LIN {X 0,Y 312.481,Z 159.56,A -85,B 0,C 180,E1 -15787.929,E2 -15787.929} C_VEL
LIN {X 0,Y 311.791,Z 159.647,A -85,B 0,C 180,E1 -15789.004,E2 -15789.004} C_VEL
LIN {X 0,Y 308.912,Z 160.004,A -85,B 0,C 180,E1 -15790.755,E2 -15790.755} C_VEL
LIN {X 0,Y 306.5,Z 160.304,A -85,B 0,C 180,E1 -15792.174,E2 -15792.174} C_VEL
LIN {X 0,Y 305.491,Z 160.433,A -85,B 0,C 180,E1 -15793.274,E2 -15793.274} C_VEL
LIN {X 0,Y 305.422,Z 160.441,A -85,B 0,C 180,E1 -15793.646,E2 -15793.646} C_VEL
LIN {X 0,Y 305.436,Z 160.44,A -85,B 0,C 180,E1 -15797.418,E2 -15797.418} C_VEL
LIN {X 0,Y 305.46,Z 160.435,A -85,B 0,C 180,E1 -15801.595,E2 -15801.595} C_VEL
LIN {X 0,Y 305.461,Z 160.432,A -85,B 0,C 180,E1 -15804.886,E2 -15804.886} C_VEL
LIN {X 0,Y 305.441,Z 160.436,A -85,B 0,C 180,E1 -15808.358,E2 -15808.358} C_VEL
LIN {X 0,Y 305.475,Z 160.43,A -85,B 0,C 180,E1 -15811.109,E2 -15811.109} C_VEL
LIN {X 0,Y 305.5,Z 160.429,A -85,B 0,C 180,E1 -15814.081,E2 -15814.081} C_VEL
LIN {X 0,Y 305.484,Z 160.426,A -85,B 0,C 180,E1 -15818.402,E2 -15818.402} C_VEL
LIN {X 0,Y 305.508,Z 160.428,A -85,B 0,C 180,E1 -15821.212,E2 -15821.212} C_VEL
LIN {X 0,Y 305.578,Z 160.412,A -85,B 0,C 180,E1 -15825.345,E2 -15825.345} C_VEL
LIN {X 0,Y 305.623,Z 160.413,A -85,B 0,C 180,E1 -15829.399,E2 -15829.399} C_VEL
LIN {X 0,Y 305.744,Z 160.396,A -85,B 0,C 180,E1 -15832.072,E2 -15832.072} C_VEL
LIN {X 0,Y 305.653,Z 160.409,A -85,B 0,C 180,E1 -15834.723,E2 -15834.723} C_VEL
LIN {X 0,Y 305.933,Z 160.373,A -85,B 0,C 180,E1 -15838.684,E2 -15838.684} C_VEL
LIN {X 0,Y 305.931,Z 160.366,A -85,B 0,C 180,E1 -15841.316,E2 -15841.316} C_VEL
LIN {X 0,Y 305.783,Z 160.392,A -85,B 0,C 180,E1 -15846.599,E2 -15846.599} C_VEL
LIN {X 0,Y 305.682,Z 160.4,A -85,B 0,C 180,E1 -15849.261,E2 -15849.261} C_VEL
LIN {X 0,Y 305.551,Z 160.423,A -85,B 0,C 180,E1 -15853.298,E2 -15853.298} C_VEL
LIN {X 0,Y 305.49,Z 160.424,A -85,B 0,C 180,E1 -15856.026,E2 -15856.026} C_VEL
LIN {X 0,Y 305.471,Z 160.432,A -85,B 0,C 180,E1 -15860.188,E2 -15860.188} C_VEL
LIN {X 0,Y 305.438,Z 160.434,A -85,B 0,C 180,E1 -15864.467,E2 -15864.467} C_VEL
LIN {X 0,Y 305.447,Z 160.437,A -85,B 0,C 180,E1 -15867.399,E2 -15867.399} C_VEL
LIN {X 0,Y 305.428,Z 160.436,A -85,B 0,C 180,E1 -15870.413,E2 -15870.413} C_VEL
LIN {X 0,Y 305.464,Z 160.429,A -85,B 0,C 180,E1 -15874.078,E2 -15874.078} C_VEL
LIN {X 0,Y 305.453,Z 160.437,A -85,B 0,C 180,E1 -15876.743,E2 -15876.743} C_VEL
LIN {X 0,Y 305.409,Z 160.442,A -85,B 0,C 180,E1 -15880.59,E2 -15880.59} C_VEL
LIN {X 0,Y 305.421,Z 160.438,A -85,B 0,C 180,E1 -15883.656,E2 -15883.656} C_VEL
LIN {X 0,Y 305.434,Z 160.436,A -85,B 0,C 180,E1 -15887.419,E2 -15887.419} C_VEL
LIN {X 0,Y 305.461,Z 160.433,A -85,B 0,C 180,E1 -15891.595,E2 -15891.595} C_VEL
LIN {X 0,Y 305.463,Z 160.437,A -85,B 0,C 180,E1 -15894.887,E2 -15894.887} C_VEL
LIN {X 0,Y 305.485,Z 160.457,A -85,B 0,C 180,E1 -15896.205,E2 -15896.205} C_VEL
LIN {X 0,Y 308.142,Z 171.998,A -85,B 0,C 180,E1 -15899.883,E2 -15899.883} C_VEL
LIN {X 0,Y 309.87,Z 180.598,A -85,B 0,C 180,E1 -15902.483,E2 -15902.483} C_VEL
LIN {X 0,Y 310.416,Z 185.1,A -85,B 0,C 180,E1 -15903.78,E2 -15903.78} C_VEL
LIN {X 0,Y 315.255,Z 212.189,A -85,B 0,C 180,E1 -15904.876,E2 -15904.876} C_VEL
LIN {X 0,Y 317.606,Z 229.16,A -85,B 0,C 180,E1 -15905.486,E2 -15905.486} C_VEL
LIN {X 0,Y 316.044,Z 293.949,A -85,B 0,C 180,E1 -15906.968,E2 -15906.968} C_VEL
LIN {X 0,Y 315.164,Z 307.123,A -85,B 0,C 180,E1 -15907.506,E2 -15907.506} C_VEL
LIN {X 0,Y 313.89,Z 320.349,A -85,B 0,C 180,E1 -15908.319,E2 -15908.319} C_VEL
LIN {X 0,Y 312.567,Z 331.466,A -85,B 0,C 180,E1 -15909.259,E2 -15909.259} C_VEL
LIN {X 0,Y 311.014,Z 343.05,A -85,B 0,C 180,E1 -15910.53,E2 -15910.53} C_VEL
LIN {X 0,Y 309.393,Z 353.483,A -85,B 0,C 180,E1 -15911.971,E2 -15911.971} C_VEL
LIN {X 0,Y 308.101,Z 362.46,A -85,B 0,C 180,E1 -15913.517,E2 -15913.517} C_VEL
LIN {X 0,Y 306.676,Z 371.281,A -85,B 0,C 180,E1 -15915.399,E2 -15915.399} C_VEL
LIN {X 0,Y 305.431,Z 378.722,A -85,B 0,C 180,E1 -15917.373,E2 -15917.373} C_VEL
LIN {X 0,Y 304.614,Z 384.707,A -85,B 0,C 180,E1 -15919.363,E2 -15919.363} C_VEL
LIN {X 0,Y 304.052,Z 389.439,A -85,B 0,C 180,E1 -15921.358,E2 -15921.358} C_VEL
LIN {X 0,Y 303.72,Z 393.058,A -85,B 0,C 180,E1 -15923.355,E2 -15923.355} C_VEL
LIN {X 0,Y 303.638,Z 394.926,A -85,B 0,C 180,E1 -15924.687,E2 -15924.687} C_VEL
LIN {X 0,Y 303.629,Z 396.329,A -85,B 0,C 180,E1 -15926.018,E2 -15926.018} C_VEL
LIN {X 0,Y 303.624,Z 397.33,A -85,B 0,C 180,E1 -15927.346,E2 -15927.346} C_VEL
LIN {X 0,Y 303.614,Z 397.94,A -85,B 0,C 180,E1 -15928.673,E2 -15928.673} C_VEL
LIN {X 0,Y 303.667,Z 398.156,A -85,B 0,C 180,E1 -15929.999,E2 -15929.999} C_VEL
LIN {X 0,Y 303.614,Z 397.933,A -85,B 0,C 180,E1 -15931.326,E2 -15931.326} C_VEL
LIN {X 0,Y 303.624,Z 397.319,A -85,B 0,C 180,E1 -15932.653,E2 -15932.653} C_VEL
LIN {X 0,Y 303.63,Z 396.314,A -85,B 0,C 180,E1 -15933.981,E2 -15933.981} C_VEL
LIN {X 0,Y 303.625,Z 394.595,A -85,B 0,C 180,E1 -15935.544,E2 -15935.544} C_VEL
LIN {X 0,Y 303.943,Z 390.715,A -85,B 0,C 180,E1 -15937.974,E2 -15937.974} C_VEL
LIN {X 0,Y 304.383,Z 386.352,A -85,B 0,C 180,E1 -15939.971,E2 -15939.971} C_VEL
LIN {X 0,Y 305.092,Z 380.8,A -85,B 0,C 180,E1 -15941.964,E2 -15941.964} C_VEL
LIN {X 0,Y 306.255,Z 373.882,A -85,B 0,C 180,E1 -15943.942,E2 -15943.942} C_VEL
LIN {X 0,Y 307.655,Z 365.226,A -85,B 0,C 180,E1 -15945.909,E2 -15945.909} C_VEL
LIN {X 0,Y 308.931,Z 356.351,A -85,B 0,C 180,E1 -15947.543,E2 -15947.543} C_VEL
LIN {X 0,Y 310.58,Z 345.437,A -85,B 0,C 180,E1 -15949.153,E2 -15949.153} C_VEL
LIN {X 0,Y 312.132,Z 334.421,A -85,B 0,C 180,E1 -15950.425,E2 -15950.425} C_VEL
LIN {X 0,Y 313.617,Z 322.074,A -85,B 0,C 180,E1 -15951.527,E2 -15951.527} C_VEL
LIN {X 0,Y 314.804,Z 310.379,A -85,B 0,C 180,E1 -15952.303,E2 -15952.303} C_VEL
LIN {X 0,Y 315.802,Z 297.871,A -85,B 0,C 180,E1 -15952.876,E2 -15952.876} C_VEL
LIN {X 0,Y 316.354,Z 281.908,A -85,B 0,C 180,E1 -15953.31,E2 -15953.31} C_VEL
LIN {X 0,Y 317.411,Z 226.976,A -85,B 0,C 180,E1 -15954.557,E2 -15954.557} C_VEL
LIN {X 0,Y 312.684,Z 197.182,A -85,B 0,C 180,E1 -15955.688,E2 -15955.688} C_VEL
LIN {X 0,Y 310.379,Z 185.064,A -85,B 0,C 180,E1 -15956.202,E2 -15956.202} C_VEL
LIN {X 0,Y 309.526,Z 178.852,A -85,B 0,C 180,E1 -15958.008,E2 -15958.008} C_VEL
LIN {X 0,Y 307.186,Z 167.923,A -85,B 0,C 180,E1 -15961.364,E2 -15961.364} C_VEL
LIN {X 0,Y 305.481,Z 160.432,A -85,B 0,C 180,E1 -15963.794,E2 -15963.794} C_VEL
LIN {X 0,Y 305.45,Z 160.429,A -85,B 0,C 180,E1 -15966.741,E2 -15966.741} C_VEL
LIN {X 0,Y 305.405,Z 160.439,A -85,B 0,C 180,E1 -15970.589,E2 -15970.589} C_VEL
LIN {X 0,Y 305.416,Z 160.441,A -85,B 0,C 180,E1 -15973.655,E2 -15973.655} C_VEL
LIN {X 0,Y 305.43,Z 160.441,A -85,B 0,C 180,E1 -15977.417,E2 -15977.417} C_VEL
LIN {X 0,Y 305.454,Z 160.435,A -85,B 0,C 180,E1 -15981.594,E2 -15981.594} C_VEL
LIN {X 0,Y 305.455,Z 160.438,A -85,B 0,C 180,E1 -15984.886,E2 -15984.886} C_VEL
LIN {X 0,Y 305.435,Z 160.435,A -85,B 0,C 180,E1 -15988.357,E2 -15988.357} C_VEL
LIN {X 0,Y 305.468,Z 160.429,A -85,B 0,C 180,E1 -15991.108,E2 -15991.108} C_VEL
LIN {X 0,Y 305.473,Z 160.431,A -85,B 0,C 180,E1 -15994.079,E2 -15994.079} C_VEL
LIN {X 0,Y 305.45,Z 160.434,A -85,B 0,C 180,E1 -15998.399,E2 -15998.399} C_VEL
LIN {X 0,Y 305.494,Z 160.429,A -85,B 0,C 180,E1 -16001.212,E2 -16001.212} C_VEL
LIN {X 0,Y 305.57,Z 160.418,A -85,B 0,C 180,E1 -16005.345,E2 -16005.345} C_VEL
LIN {X 0,Y 305.614,Z 160.411,A -85,B 0,C 180,E1 -16009.399,E2 -16009.399} C_VEL
LIN {X 0,Y 305.729,Z 160.4,A -85,B 0,C 180,E1 -16012.072,E2 -16012.072} C_VEL
LIN {X 0,Y 305.645,Z 160.41,A -85,B 0,C 180,E1 -16014.723,E2 -16014.723} C_VEL
LIN {X 0,Y 305.924,Z 160.373,A -85,B 0,C 180,E1 -16018.684,E2 -16018.684} C_VEL
LIN {X 0,Y 305.926,Z 160.376,A -85,B 0,C 180,E1 -16021.316,E2 -16021.316} C_VEL
LIN {X 0,Y 305.777,Z 160.392,A -85,B 0,C 180,E1 -16026.599,E2 -16026.599} C_VEL
LIN {X 0,Y 305.686,Z 160.407,A -85,B 0,C 180,E1 -16029.261,E2 -16029.261} C_VEL
LIN {X 0,Y 305.563,Z 160.416,A -85,B 0,C 180,E1 -16033.297,E2 -16033.297} C_VEL
LIN {X 0,Y 305.505,Z 160.429,A -85,B 0,C 180,E1 -16036.025,E2 -16036.025} C_VEL
LIN {X 0,Y 305.478,Z 160.428,A -85,B 0,C 180,E1 -16040.188,E2 -16040.188} C_VEL
LIN {X 0,Y 305.479,Z 160.433,A -85,B 0,C 180,E1 -16043.04,E2 -16043.04} C_VEL
LIN {X 0,Y 305.446,Z 160.43,A -85,B 0,C 180,E1 -16046.191,E2 -16046.191} C_VEL
LIN {X 0,Y 305.442,Z 160.439,A -85,B 0,C 180,E1 -16049.034,E2 -16049.034} C_VEL
LIN {X 0,Y 305.43,Z 160.434,A -85,B 0,C 180,E1 -16051.954,E2 -16051.954} C_VEL
LIN {X 0,Y 305.455,Z 160.437,A -85,B 0,C 180,E1 -16055.114,E2 -16055.114} C_VEL
LIN {X 0,Y 305.427,Z 160.439,A -85,B 0,C 180,E1 -16058.526,E2 -16058.526} C_VEL
LIN {X 0,Y 305.431,Z 160.44,A -85,B 0,C 180,E1 -16062.583,E2 -16062.583} C_VEL
LIN {X 0,Y 305.418,Z 160.439,A -85,B 0,C 180,E1 -16066.345,E2 -16066.345} C_VEL
LIN {X 0,Y 305.454,Z 160.435,A -85,B 0,C 180,E1 -16069.893,E2 -16069.893} C_VEL
LIN {X 0,Y 305.46,Z 160.434,A -85,B 0,C 180,E1 -16073.637,E2 -16073.637} C_VEL
LIN {X 0,Y 305.463,Z 160.438,A -85,B 0,C 180,E1 -16076.484,E2 -16076.484} C_VEL
LIN {X 0,Y 305.429,Z 160.437,A -85,B 0,C 180,E1 -16079.589,E2 -16079.589} C_VEL
LIN {X 0,Y 305.527,Z 160.543,A -85,B 0,C 180,E1 -16081.912,E2 -16081.912} C_VEL
LIN {X 0,Y 306.578,Z 165.2,A -85,B 0,C 180,E1 -16083.493,E2 -16083.493} C_VEL
LIN {X 0,Y 314.759,Z 184.793,A -85,B 0,C 180,E1 -16084.743,E2 -16084.743} C_VEL
LIN {X 0,Y 317.517,Z 192.242,A -85,B 0,C 180,E1 -16085.163,E2 -16085.163} C_VEL
LIN {X 0,Y 318.252,Z 196.661,A -85,B 0,C 180,E1 -16085.333,E2 -16085.333} C_VEL
LIN {X 0,Y 316.461,Z 271.983,A -85,B 0,C 180,E1 -16087.045,E2 -16087.045} C_VEL
LIN {X 0,Y 315.766,Z 285.365,A -85,B 0,C 180,E1 -16087.596,E2 -16087.596} C_VEL
LIN {X 0,Y 314.898,Z 296.992,A -85,B 0,C 180,E1 -16088.307,E2 -16088.307} C_VEL
LIN {X 0,Y 313.577,Z 309.444,A -85,B 0,C 180,E1 -16089.33,E2 -16089.33} C_VEL
LIN {X 0,Y 312.107,Z 321.083,A -85,B 0,C 180,E1 -16090.603,E2 -16090.603} C_VEL
LIN {X 0,Y 310.863,Z 331.53,A -85,B 0,C 180,E1 -16092.063,E2 -16092.063} C_VEL
LIN {X 0,Y 309.504,Z 340.047,A -85,B 0,C 180,E1 -16093.511,E2 -16093.511} C_VEL
LIN {X 0,Y 308.172,Z 347.905,A -85,B 0,C 180,E1 -16095.135,E2 -16095.135} C_VEL
LIN {X 0,Y 306.815,Z 355.583,A -85,B 0,C 180,E1 -16097.096,E2 -16097.096} C_VEL
LIN {X 0,Y 305.606,Z 362.627,A -85,B 0,C 180,E1 -16099.399,E2 -16099.399} C_VEL
LIN {X 0,Y 304.855,Z 367.315,A -85,B 0,C 180,E1 -16101.383,E2 -16101.383} C_VEL
LIN {X 0,Y 304.369,Z 370.9,A -85,B 0,C 180,E1 -16103.371,E2 -16103.371} C_VEL
LIN {X 0,Y 304.151,Z 372.752,A -85,B 0,C 180,E1 -16104.697,E2 -16104.697} C_VEL
LIN {X 0,Y 303.94,Z 374.146,A -85,B 0,C 180,E1 -16106.023,E2 -16106.023} C_VEL
LIN {X 0,Y 303.684,Z 375.749,A -85,B 0,C 180,E1 -16108.675,E2 -16108.675} C_VEL
LIN {X 0,Y 303.678,Z 375.979,A -85,B 0,C 180,E1 -16110.001,E2 -16110.001} C_VEL
LIN {X 0,Y 303.683,Z 375.788,A -85,B 0,C 180,E1 -16111.327,E2 -16111.327} C_VEL
LIN {X 0,Y 303.934,Z 374.237,A -85,B 0,C 180,E1 -16113.978,E2 -16113.978} C_VEL
LIN {X 0,Y 304.128,Z 372.883,A -85,B 0,C 180,E1 -16115.304,E2 -16115.304} C_VEL
LIN {X 0,Y 304.472,Z 370.494,A -85,B 0,C 180,E1 -16116.995,E2 -16116.995} C_VEL
LIN {X 0,Y 305.006,Z 366.145,A -85,B 0,C 180,E1 -16119.283,E2 -16119.283} C_VEL
LIN {X 0,Y 305.917,Z 361.133,A -85,B 0,C 180,E1 -16121.261,E2 -16121.261} C_VEL
LIN {X 0,Y 306.998,Z 354.824,A -85,B 0,C 180,E1 -16123.234,E2 -16123.234} C_VEL
LIN {X 0,Y 308.313,Z 346.926,A -85,B 0,C 180,E1 -16125.198,E2 -16125.198} C_VEL
LIN {X 0,Y 310.034,Z 337.093,A -85,B 0,C 180,E1 -16127.139,E2 -16127.139} C_VEL
LIN {X 0,Y 311.47,Z 326.779,A -85,B 0,C 180,E1 -16128.756,E2 -16128.756} C_VEL
LIN {X 0,Y 312.826,Z 316.549,A -85,B 0,C 180,E1 -16130.036,E2 -16130.036} C_VEL
LIN {X 0,Y 314.139,Z 305.354,A -85,B 0,C 180,E1 -16131.147,E2 -16131.147} C_VEL
LIN {X 0,Y 315.314,Z 292.729,A -85,B 0,C 180,E1 -16132.094,E2 -16132.094} C_VEL
LIN {X 0,Y 316.136,Z 280.065,A -85,B 0,C 180,E1 -16132.766,E2 -16132.766} C_VEL
LIN {X 0,Y 316.79,Z 267.014,A -85,B 0,C 180,E1 -16133.191,E2 -16133.191} C_VEL
LIN {X 0,Y 318.32,Z 196.121,A -85,B 0,C 180,E1 -16134.791,E2 -16134.791} C_VEL
LIN {X 0,Y 316.871,Z 190.339,A -85,B 0,C 180,E1 -16135.055,E2 -16135.055} C_VEL
LIN {X 0,Y 309.139,Z 171.149,A -85,B 0,C 180,E1 -16136.221,E2 -16136.221} C_VEL
LIN {X 0,Y 306.606,Z 165.204,A -85,B 0,C 180,E1 -16136.625,E2 -16136.625} C_VEL
LIN {X 0,Y 305.495,Z 160.433,A -85,B 0,C 180,E1 -16138.326,E2 -16138.326} C_VEL
LIN {X 0,Y 305.439,Z 160.435,A -85,B 0,C 180,E1 -16141.953,E2 -16141.953} C_VEL
LIN {X 0,Y 305.464,Z 160.434,A -85,B 0,C 180,E1 -16145.113,E2 -16145.113} C_VEL
LIN {X 0,Y 305.421,Z 160.438,A -85,B 0,C 180,E1 -16148.522,E2 -16148.522} C_VEL
LIN {X 0,Y 305.436,Z 160.437,A -85,B 0,C 180,E1 -16152.582,E2 -16152.582} C_VEL
LIN {X 0,Y 305.422,Z 160.441,A -85,B 0,C 180,E1 -16153.646,E2 -16153.646} C_VEL
LIN {X 0,Y 304.783,Z 160.528,A -85,B 0,C 180,E1 -16154.746,E2 -16154.746} C_VEL
LIN {X 0,Y 301.917,Z 160.887,A -85,B 0,C 180,E1 -16156.535,E2 -16156.535} C_VEL
LIN {X 0,Y 299.467,Z 161.186,A -85,B 0,C 180,E1 -16157.987,E2 -16157.987} C_VEL
LIN {X 0,Y 298.416,Z 161.311,A -85,B 0,C 180,E1 -16159.113,E2 -16159.113} C_VEL
LIN {X 0,Y 298.332,Z 161.318,A -85,B 0,C 180,E1 -16159.494,E2 -16159.494} C_VEL
LIN {X 0,Y 298.427,Z 161.311,A -85,B 0,C 180,E1 -16163.197,E2 -16163.197} C_VEL
LIN {X 0,Y 298.393,Z 161.317,A -85,B 0,C 180,E1 -16167.199,E2 -16167.199} C_VEL
LIN {X 0,Y 298.402,Z 161.31,A -85,B 0,C 180,E1 -16170.625,E2 -16170.625} C_VEL
LIN {X 0,Y 298.445,Z 161.309,A -85,B 0,C 180,E1 -16174.92,E2 -16174.92} C_VEL
LIN {X 0,Y 298.42,Z 161.303,A -85,B 0,C 180,E1 -16177.864,E2 -16177.864} C_VEL
LIN {X 0,Y 298.473,Z 161.308,A -85,B 0,C 180,E1 -16180.752,E2 -16180.752} C_VEL
LIN {X 0,Y 298.509,Z 161.293,A -85,B 0,C 180,E1 -16184.99,E2 -16184.99} C_VEL
LIN {X 0,Y 298.581,Z 161.29,A -85,B 0,C 180,E1 -16189.146,E2 -16189.146} C_VEL
LIN {X 0,Y 298.696,Z 161.274,A -85,B 0,C 180,E1 -16191.884,E2 -16191.884} C_VEL
LIN {X 0,Y 298.623,Z 161.285,A -85,B 0,C 180,E1 -16194.598,E2 -16194.598} C_VEL
LIN {X 0,Y 298.901,Z 161.249,A -85,B 0,C 180,E1 -16198.653,E2 -16198.653} C_VEL
LIN {X 0,Y 298.899,Z 161.242,A -85,B 0,C 180,E1 -16201.347,E2 -16201.347} C_VEL
LIN {X 0,Y 298.731,Z 161.27,A -85,B 0,C 180,E1 -16206.755,E2 -16206.755} C_VEL
LIN {X 0,Y 298.614,Z 161.28,A -85,B 0,C 180,E1 -16209.483,E2 -16209.483} C_VEL
LIN {X 0,Y 298.506,Z 161.303,A -85,B 0,C 180,E1 -16213.618,E2 -16213.618} C_VEL
LIN {X 0,Y 298.428,Z 161.301,A -85,B 0,C 180,E1 -16216.416,E2 -16216.416} C_VEL
LIN {X 0,Y 298.427,Z 161.313,A -85,B 0,C 180,E1 -16219.609,E2 -16219.609} C_VEL
LIN {X 0,Y 298.381,Z 161.313,A -85,B 0,C 180,E1 -16223.604,E2 -16223.604} C_VEL
LIN {X 0,Y 298.401,Z 161.313,A -85,B 0,C 180,E1 -16226.583,E2 -16226.583} C_VEL
LIN {X 0,Y 298.391,Z 161.314,A -85,B 0,C 180,E1 -16229.644,E2 -16229.644} C_VEL
LIN {X 0,Y 298.392,Z 161.316,A -85,B 0,C 180,E1 -16232.801,E2 -16232.801} C_VEL
LIN {X 0,Y 298.427,Z 161.313,A -85,B 0,C 180,E1 -16236.802,E2 -16236.802} C_VEL
LIN {X 0,Y 298.373,Z 161.318,A -85,B 0,C 180,E1 -16239.492,E2 -16239.492} C_VEL
LIN {X 0,Y 298.37,Z 161.32,A -85,B 0,C 180,E1 -16243.097,E2 -16243.097} C_VEL
LIN {X 0,Y 298.37,Z 161.318,A -85,B 0,C 180,E1 -16246.915,E2 -16246.915} C_VEL
LIN {X 0,Y 298.385,Z 161.316,A -85,B 0,C 180,E1 -16251.011,E2 -16251.011} C_VEL
LIN {X 0,Y 298.406,Z 161.314,A -85,B 0,C 180,E1 -16253.928,E2 -16253.928} C_VEL
LIN {X 0,Y 298.463,Z 161.508,A -85,B 0,C 180,E1 -16255.716,E2 -16255.716} C_VEL
LIN {X 0,Y 300.842,Z 171.699,A -85,B 0,C 180,E1 -16259.073,E2 -16259.073} C_VEL
LIN {X 0,Y 302.701,Z 180.807,A -85,B 0,C 180,E1 -16261.918,E2 -16261.918} C_VEL
LIN {X 0,Y 303.392,Z 184.77,A -85,B 0,C 180,E1 -16263.115,E2 -16263.115} C_VEL
LIN {X 0,Y 305.029,Z 191.285,A -85,B 0,C 180,E1 -16263.445,E2 -16263.445} C_VEL
LIN {X 0,Y 309.487,Z 217.498,A -85,B 0,C 180,E1 -16264.513,E2 -16264.513} C_VEL
LIN {X 0,Y 311.149,Z 229.779,A -85,B 0,C 180,E1 -16264.964,E2 -16264.964} C_VEL
LIN {X 0,Y 309.542,Z 293.704,A -85,B 0,C 180,E1 -16266.455,E2 -16266.455} C_VEL
LIN {X 0,Y 308.564,Z 307.636,A -85,B 0,C 180,E1 -16267.042,E2 -16267.042} C_VEL
LIN {X 0,Y 307.286,Z 320.096,A -85,B 0,C 180,E1 -16267.828,E2 -16267.828} C_VEL
LIN {X 0,Y 305.932,Z 331.211,A -85,B 0,C 180,E1 -16268.788,E2 -16268.788} C_VEL
LIN {X 0,Y 304.305,Z 342.794,A -85,B 0,C 180,E1 -16270.083,E2 -16270.083} C_VEL
LIN {X 0,Y 302.61,Z 353.225,A -85,B 0,C 180,E1 -16271.552,E2 -16271.552} C_VEL
LIN {X 0,Y 301.147,Z 362.926,A -85,B 0,C 180,E1 -16273.278,E2 -16273.278} C_VEL
LIN {X 0,Y 299.761,Z 371.022,A -85,B 0,C 180,E1 -16275.054,E2 -16275.054} C_VEL
LIN {X 0,Y 298.487,Z 378.464,A -85,B 0,C 180,E1 -16277.074,E2 -16277.074} C_VEL
LIN {X 0,Y 297.614,Z 384.448,A -85,B 0,C 180,E1 -16279.11,E2 -16279.11} C_VEL
LIN {X 0,Y 297.008,Z 389.18,A -85,B 0,C 180,E1 -16281.152,E2 -16281.152} C_VEL
LIN {X 0,Y 296.645,Z 392.799,A -85,B 0,C 180,E1 -16283.196,E2 -16283.196} C_VEL
LIN {X 0,Y 296.552,Z 394.667,A -85,B 0,C 180,E1 -16284.56,E2 -16284.56} C_VEL
LIN {X 0,Y 296.527,Z 396.07,A -85,B 0,C 180,E1 -16285.922,E2 -16285.922} C_VEL
LIN {X 0,Y 296.548,Z 397.072,A -85,B 0,C 180,E1 -16287.283,E2 -16287.283} C_VEL
LIN {X 0,Y 296.531,Z 397.682,A -85,B 0,C 180,E1 -16288.641,E2 -16288.641} C_VEL
LIN {X 0,Y 296.579,Z 397.898,A -85,B 0,C 180,E1 -16289.999,E2 -16289.999} C_VEL
LIN {X 0,Y 296.531,Z 397.674,A -85,B 0,C 180,E1 -16291.357,E2 -16291.357} C_VEL
LIN {X 0,Y 296.549,Z 397.06,A -85,B 0,C 180,E1 -16292.716,E2 -16292.716} C_VEL
LIN {X 0,Y 296.527,Z 396.054,A -85,B 0,C 180,E1 -16294.077,E2 -16294.077} C_VEL
LIN {X 0,Y 296.546,Z 394.558,A -85,B 0,C 180,E1 -16295.508,E2 -16295.508} C_VEL
LIN {X 0,Y 296.782,Z 391.689,A -85,B 0,C 180,E1 -16297.483,E2 -16297.483} C_VEL
LIN {X 0,Y 297.19,Z 387.693,A -85,B 0,C 180,E1 -16299.528,E2 -16299.528} C_VEL
LIN {X 0,Y 297.957,Z 381.553,A -85,B 0,C 180,E1 -16301.91,E2 -16301.91} C_VEL
LIN {X 0,Y 299.106,Z 374.858,A -85,B 0,C 180,E1 -16303.935,E2 -16303.935} C_VEL
LIN {X 0,Y 300.535,Z 366.557,A -85,B 0,C 180,E1 -16305.948,E2 -16305.948} C_VEL
LIN {X 0,Y 301.85,Z 358.043,A -85,B 0,C 180,E1 -16307.618,E2 -16307.618} C_VEL
LIN {X 0,Y 303.475,Z 347.531,A -85,B 0,C 180,E1 -16309.268,E2 -16309.268} C_VEL
LIN {X 0,Y 305.275,Z 335.707,A -85,B 0,C 180,E1 -16310.729,E2 -16310.729} C_VEL
LIN {X 0,Y 306.796,Z 323.801,A -85,B 0,C 180,E1 -16311.853,E2 -16311.853} C_VEL
LIN {X 0,Y 308.123,Z 311.414,A -85,B 0,C 180,E1 -16312.725,E2 -16312.725} C_VEL
LIN {X 0,Y 309.218,Z 298.669,A -85,B 0,C 180,E1 -16313.347,E2 -16313.347} C_VEL
LIN {X 0,Y 309.786,Z 285.21,A -85,B 0,C 180,E1 -16313.745,E2 -16313.745} C_VEL
LIN {X 0,Y 310.961,Z 228.075,A -85,B 0,C 180,E1 -16315.067,E2 -16315.067} C_VEL
LIN {X 0,Y 306.443,Z 199.125,A -85,B 0,C 180,E1 -16316.194,E2 -16316.194} C_VEL
LIN {X 0,Y 303.978,Z 186.837,A -85,B 0,C 180,E1 -16316.738,E2 -16316.738} C_VEL
LIN {X 0,Y 303.38,Z 184.674,A -85,B 0,C 180,E1 -16316.884,E2 -16316.884} C_VEL
LIN {X 0,Y 301.58,Z 175.207,A -85,B 0,C 180,E1 -16319.785,E2 -16319.785} C_VEL
LIN {X 0,Y 298.973,Z 163.637,A -85,B 0,C 180,E1 -16323.532,E2 -16323.532} C_VEL
LIN {X 0,Y 298.423,Z 161.31,A -85,B 0,C 180,E1 -16324.363,E2 -16324.363} C_VEL
LIN {X 0,Y 298.394,Z 161.309,A -85,B 0,C 180,E1 -16327.76,E2 -16327.76} C_VEL
LIN {X 0,Y 298.343,Z 161.321,A -85,B 0,C 180,E1 -16331.267,E2 -16331.267} C_VEL
LIN {X 0,Y 298.35,Z 161.323,A -85,B 0,C 180,E1 -16335.034,E2 -16335.034} C_VEL
LIN {X 0,Y 298.343,Z 161.323,A -85,B 0,C 180,E1 -16338.92,E2 -16338.92} C_VEL
LIN {X 0,Y 298.391,Z 161.314,A -85,B 0,C 180,E1 -16342.238,E2 -16342.238} C_VEL
LIN {X 0,Y 298.401,Z 161.312,A -85,B 0,C 180,E1 -16345.58,E2 -16345.58} C_VEL
LIN {X 0,Y 298.37,Z 161.319,A -85,B 0,C 180,E1 -16348.788,E2 -16348.788} C_VEL
LIN {X 0,Y 298.403,Z 161.306,A -85,B 0,C 180,E1 -16351.898,E2 -16351.898} C_VEL
LIN {X 0,Y 298.406,Z 161.313,A -85,B 0,C 180,E1 -16354.917,E2 -16354.917} C_VEL
LIN {X 0,Y 298.382,Z 161.31,A -85,B 0,C 180,E1 -16357.861,E2 -16357.861} C_VEL
LIN {X 0,Y 298.445,Z 161.309,A -85,B 0,C 180,E1 -16360.751,E2 -16360.751} C_VEL
LIN {X 0,Y 298.502,Z 161.3,A -85,B 0,C 180,E1 -16364.99,E2 -16364.99} C_VEL
LIN {X 0,Y 298.572,Z 161.287,A -85,B 0,C 180,E1 -16369.146,E2 -16369.146} C_VEL
LIN {X 0,Y 298.675,Z 161.277,A -85,B 0,C 180,E1 -16371.884,E2 -16371.884} C_VEL
LIN {X 0,Y 298.616,Z 161.286,A -85,B 0,C 180,E1 -16374.598,E2 -16374.598} C_VEL
LIN {X 0,Y 298.892,Z 161.249,A -85,B 0,C 180,E1 -16378.653,E2 -16378.653} C_VEL
LIN {X 0,Y 298.894,Z 161.252,A -85,B 0,C 180,E1 -16381.347,E2 -16381.347} C_VEL
LIN {X 0,Y 298.726,Z 161.27,A -85,B 0,C 180,E1 -16386.756,E2 -16386.756} C_VEL
LIN {X 0,Y 298.618,Z 161.289,A -85,B 0,C 180,E1 -16389.483,E2 -16389.483} C_VEL
LIN {X 0,Y 298.515,Z 161.297,A -85,B 0,C 180,E1 -16393.617,E2 -16393.617} C_VEL
LIN {X 0,Y 298.446,Z 161.307,A -85,B 0,C 180,E1 -16396.415,E2 -16396.415} C_VEL
LIN {X 0,Y 298.436,Z 161.305,A -85,B 0,C 180,E1 -16399.618,E2 -16399.618} C_VEL
LIN {X 0,Y 298.405,Z 161.314,A -85,B 0,C 180,E1 -16403.602,E2 -16403.602} C_VEL
LIN {X 0,Y 298.396,Z 161.309,A -85,B 0,C 180,E1 -16406.584,E2 -16406.584} C_VEL
LIN {X 0,Y 298.387,Z 161.315,A -85,B 0,C 180,E1 -16409.645,E2 -16409.645} C_VEL
LIN {X 0,Y 298.387,Z 161.314,A -85,B 0,C 180,E1 -16412.801,E2 -16412.801} C_VEL
LIN {X 0,Y 298.421,Z 161.314,A -85,B 0,C 180,E1 -16416.803,E2 -16416.803} C_VEL
LIN {X 0,Y 298.368,Z 161.317,A -85,B 0,C 180,E1 -16419.493,E2 -16419.493} C_VEL
LIN {X 0,Y 298.366,Z 161.319,A -85,B 0,C 180,E1 -16423.099,E2 -16423.099} C_VEL
LIN {X 0,Y 298.37,Z 161.319,A -85,B 0,C 180,E1 -16426.917,E2 -16426.917} C_VEL
LIN {X 0,Y 298.392,Z 161.314,A -85,B 0,C 180,E1 -16431.01,E2 -16431.01} C_VEL
LIN {X 0,Y 298.403,Z 161.314,A -85,B 0,C 180,E1 -16433.93,E2 -16433.93} C_VEL
LIN {X 0,Y 298.391,Z 161.315,A -85,B 0,C 180,E1 -16437.201,E2 -16437.201} C_VEL
LIN {X 0,Y 298.471,Z 161.411,A -85,B 0,C 180,E1 -16441.379,E2 -16441.379} C_VEL
LIN {X 0,Y 299.467,Z 165.684,A -85,B 0,C 180,E1 -16442.832,E2 -16442.832} C_VEL
LIN {X 0,Y 307.39,Z 184.115,A -85,B 0,C 180,E1 -16444.068,E2 -16444.068} C_VEL
LIN {X 0,Y 311.452,Z 195.204,A -85,B 0,C 180,E1 -16444.713,E2 -16444.713} C_VEL
LIN {X 0,Y 311.819,Z 198.379,A -85,B 0,C 180,E1 -16444.825,E2 -16444.825} C_VEL
LIN {X 0,Y 309.954,Z 272.259,A -85,B 0,C 180,E1 -16446.534,E2 -16446.534} C_VEL
LIN {X 0,Y 309.224,Z 285.634,A -85,B 0,C 180,E1 -16447.095,E2 -16447.095} C_VEL
LIN {X 0,Y 308.316,Z 297.259,A -85,B 0,C 180,E1 -16447.82,E2 -16447.82} C_VEL
LIN {X 0,Y 306.967,Z 309.708,A -85,B 0,C 180,E1 -16448.864,E2 -16448.864} C_VEL
LIN {X 0,Y 305.442,Z 321.346,A -85,B 0,C 180,E1 -16450.162,E2 -16450.162} C_VEL
LIN {X 0,Y 304.062,Z 332.151,A -85,B 0,C 180,E1 -16451.706,E2 -16451.706} C_VEL
LIN {X 0,Y 302.434,Z 341.998,A -85,B 0,C 180,E1 -16453.462,E2 -16453.462} C_VEL
LIN {X 0,Y 300.792,Z 350.9,A -85,B 0,C 180,E1 -16455.454,E2 -16455.454} C_VEL
LIN {X 0,Y 299.524,Z 358.06,A -85,B 0,C 180,E1 -16457.466,E2 -16457.466} C_VEL
LIN {X 0,Y 298.641,Z 362.887,A -85,B 0,C 180,E1 -16459.149,E2 -16459.149} C_VEL
LIN {X 0,Y 297.822,Z 367.576,A -85,B 0,C 180,E1 -16461.178,E2 -16461.178} C_VEL
LIN {X 0,Y 297.307,Z 371.161,A -85,B 0,C 180,E1 -16463.213,E2 -16463.213} C_VEL
LIN {X 0,Y 297.087,Z 373.011,A -85,B 0,C 180,E1 -16464.571,E2 -16464.571} C_VEL
LIN {X 0,Y 296.881,Z 374.405,A -85,B 0,C 180,E1 -16465.928,E2 -16465.928} C_VEL
LIN {X 0,Y 296.6,Z 376.008,A -85,B 0,C 180,E1 -16468.643,E2 -16468.643} C_VEL
LIN {X 0,Y 296.59,Z 376.238,A -85,B 0,C 180,E1 -16470.001,E2 -16470.001} C_VEL
LIN {X 0,Y 296.6,Z 376.047,A -85,B 0,C 180,E1 -16471.358,E2 -16471.358} C_VEL
LIN {X 0,Y 296.874,Z 374.495,A -85,B 0,C 180,E1 -16474.073,E2 -16474.073} C_VEL
LIN {X 0,Y 297.066,Z 373.141,A -85,B 0,C 180,E1 -16475.431,E2 -16475.431} C_VEL
LIN {X 0,Y 297.459,Z 370.386,A -85,B 0,C 180,E1 -16477.399,E2 -16477.399} C_VEL
LIN {X 0,Y 297.997,Z 366.403,A -85,B 0,C 180,E1 -16479.503,E2 -16479.503} C_VEL
LIN {X 0,Y 298.966,Z 361.39,A -85,B 0,C 180,E1 -16481.527,E2 -16481.527} C_VEL
LIN {X 0,Y 300.094,Z 355.081,A -85,B 0,C 180,E1 -16483.545,E2 -16483.545} C_VEL
LIN {X 0,Y 301.475,Z 347.182,A -85,B 0,C 180,E1 -16485.551,E2 -16485.551} C_VEL
LIN {X 0,Y 303.256,Z 337.349,A -85,B 0,C 180,E1 -16487.535,E2 -16487.535} C_VEL
LIN {X 0,Y 304.757,Z 327.03,A -85,B 0,C 180,E1 -16489.185,E2 -16489.185} C_VEL
LIN {X 0,Y 306.185,Z 316.802,A -85,B 0,C 180,E1 -16490.49,E2 -16490.49} C_VEL
LIN {X 0,Y 307.551,Z 305.606,A -85,B 0,C 180,E1 -16491.622,E2 -16491.622} C_VEL
LIN {X 0,Y 308.752,Z 292.979,A -85,B 0,C 180,E1 -16492.589,E2 -16492.589} C_VEL
LIN {X 0,Y 309.614,Z 280.311,A -85,B 0,C 180,E1 -16493.273,E2 -16493.273} C_VEL
LIN {X 0,Y 310.291,Z 267.253,A -85,B 0,C 180,E1 -16493.706,E2 -16493.706} C_VEL
LIN {X 0,Y 311.872,Z 197.115,A -85,B 0,C 180,E1 -16495.32,E2 -16495.32} C_VEL
LIN {X 0,Y 310.588,Z 192.464,A -85,B 0,C 180,E1 -16495.551,E2 -16495.551} C_VEL
LIN {X 0,Y 303.48,Z 174.735,A -85,B 0,C 180,E1 -16496.66,E2 -16496.66} C_VEL
LIN {X 0,Y 299.402,Z 165.465,A -85,B 0,C 180,E1 -16497.325,E2 -16497.325} C_VEL
LIN {X 0,Y 298.457,Z 161.309,A -85,B 0,C 180,E1 -16498.816,E2 -16498.816} C_VEL
LIN {X 0,Y 298.395,Z 161.314,A -85,B 0,C 180,E1 -16502.801,E2 -16502.801} C_VEL
LIN {X 0,Y 298.428,Z 161.309,A -85,B 0,C 180,E1 -16506.802,E2 -16506.802} C_VEL
LIN {X 0,Y 298.349,Z 161.323,A -85,B 0,C 180,E1 -16511.268,E2 -16511.268} C_VEL
LIN {X 0,Y 298.355,Z 161.321,A -85,B 0,C 180,E1 -16515.035,E2 -16515.035} C_VEL
LIN {X 0,Y 298.349,Z 161.321,A -85,B 0,C 180,E1 -16518.921,E2 -16518.921} C_VEL
LIN {X 0,Y 298.332,Z 161.318,A -85,B 0,C 180,E1 -16519.494,E2 -16519.494} C_VEL
LIN {X 0,Y 297.68,Z 161.4,A -85,B 0,C 180,E1 -16520.621,E2 -16520.621} C_VEL
LIN {X 0,Y 294.875,Z 161.752,A -85,B 0,C 180,E1 -16522.457,E2 -16522.457} C_VEL
LIN {X 0,Y 292.483,Z 162.049,A -85,B 0,C 180,E1 -16523.947,E2 -16523.947} C_VEL
LIN {X 0,Y 291.439,Z 162.177,A -85,B 0,C 180,E1 -16525.1,E2 -16525.1} C_VEL
LIN {X 0,Y 291.346,Z 162.187,A -85,B 0,C 180,E1 -16525.491,E2 -16525.491} C_VEL
LIN {X 0,Y 291.366,Z 162.189,A -85,B 0,C 180,E1 -16527.95,E2 -16527.95} C_VEL
LIN {X 0,Y 291.344,Z 162.189,A -85,B 0,C 180,E1 -16531.154,E2 -16531.154} C_VEL
LIN {X 0,Y 291.362,Z 162.191,A -85,B 0,C 180,E1 -16534.267,E2 -16534.267} C_VEL
LIN {X 0,Y 291.373,Z 162.181,A -85,B 0,C 180,E1 -16537.299,E2 -16537.299} C_VEL
LIN {X 0,Y 291.404,Z 162.185,A -85,B 0,C 180,E1 -16540.266,E2 -16540.266} C_VEL
LIN {X 0,Y 291.473,Z 162.169,A -85,B 0,C 180,E1 -16544.682,E2 -16544.682} C_VEL
LIN {X 0,Y 291.526,Z 162.17,A -85,B 0,C 180,E1 -16548.88,E2 -16548.88} C_VEL
LIN {X 0,Y 291.65,Z 162.151,A -85,B 0,C 180,E1 -16551.687,E2 -16551.687} C_VEL
LIN {X 0,Y 291.593,Z 162.159,A -85,B 0,C 180,E1 -16554.468,E2 -16554.468} C_VEL
LIN {X 0,Y 291.868,Z 162.125,A -85,B 0,C 180,E1 -16558.62,E2 -16558.62} C_VEL
LIN {X 0,Y 291.867,Z 162.117,A -85,B 0,C 180,E1 -16561.38,E2 -16561.38} C_VEL
LIN {X 0,Y 291.682,Z 162.148,A -85,B 0,C 180,E1 -16566.919,E2 -16566.919} C_VEL
LIN {X 0,Y 291.56,Z 162.158,A -85,B 0,C 180,E1 -16569.714,E2 -16569.714} C_VEL
LIN {X 0,Y 291.469,Z 162.177,A -85,B 0,C 180,E1 -16573.953,E2 -16573.953} C_VEL
LIN {X 0,Y 291.38,Z 162.178,A -85,B 0,C 180,E1 -16576.824,E2 -16576.824} C_VEL
LIN {X 0,Y 291.391,Z 162.188,A -85,B 0,C 180,E1 -16579.842,E2 -16579.842} C_VEL
LIN {X 0,Y 291.325,Z 162.191,A -85,B 0,C 180,E1 -16584.212,E2 -16584.212} C_VEL
LIN {X 0,Y 291.349,Z 162.193,A -85,B 0,C 180,E1 -16587.279,E2 -16587.279} C_VEL
LIN {X 0,Y 291.317,Z 162.194,A -85,B 0,C 180,E1 -16590.439,E2 -16590.439} C_VEL
LIN {X 0,Y 291.343,Z 162.189,A -85,B 0,C 180,E1 -16593.699,E2 -16593.699} C_VEL
LIN {X 0,Y 291.358,Z 162.189,A -85,B 0,C 180,E1 -16597.249,E2 -16597.249} C_VEL
LIN {X 0,Y 291.3,Z 162.201,A -85,B 0,C 180,E1 -16600.648,E2 -16600.648} C_VEL
LIN {X 0,Y 291.282,Z 162.201,A -85,B 0,C 180,E1 -16604.404,E2 -16604.404} C_VEL
LIN {X 0,Y 291.295,Z 162.2,A -85,B 0,C 180,E1 -16608.412,E2 -16608.412} C_VEL
LIN {X 0,Y 291.335,Z 162.193,A -85,B 0,C 180,E1 -16611.155,E2 -16611.155} C_VEL
LIN {X 0,Y 291.356,Z 162.195,A -85,B 0,C 180,E1 -16614.625,E2 -16614.625} C_VEL
LIN {X 0,Y 291.387,Z 162.233,A -85,B 0,C 180,E1 -16615.09,E2 -16615.09} C_VEL
LIN {X 0,Y 293.552,Z 171.399,A -85,B 0,C 180,E1 -16618.216,E2 -16618.216} C_VEL
LIN {X 0,Y 295.751,Z 181.96,A -85,B 0,C 180,E1 -16621.623,E2 -16621.623} C_VEL
LIN {X 0,Y 296.204,Z 184.467,A -85,B 0,C 180,E1 -16622.403,E2 -16622.403} C_VEL
LIN {X 0,Y 298.324,Z 190.602,A -85,B 0,C 180,E1 -16622.788,E2 -16622.788} C_VEL
LIN {X 0,Y 302.826,Z 216.807,A -85,B 0,C 180,E1 -16623.899,E2 -16623.899} C_VEL
LIN {X 0,Y 304.683,Z 230.691,A -85,B 0,C 180,E1 -16624.424,E2 -16624.424} C_VEL
LIN {X 0,Y 303.056,Z 293.459,A -85,B 0,C 180,E1 -16625.92,E2 -16625.92} C_VEL
LIN {X 0,Y 302.049,Z 307.387,A -85,B 0,C 180,E1 -16626.518,E2 -16626.518} C_VEL
LIN {X 0,Y 300.716,Z 319.842,A -85,B 0,C 180,E1 -16627.317,E2 -16627.317} C_VEL
LIN {X 0,Y 299.305,Z 330.956,A -85,B 0,C 180,E1 -16628.295,E2 -16628.295} C_VEL
LIN {X 0,Y 297.614,Z 342.537,A -85,B 0,C 180,E1 -16629.615,E2 -16629.615} C_VEL
LIN {X 0,Y 295.864,Z 352.969,A -85,B 0,C 180,E1 -16631.116,E2 -16631.116} C_VEL
LIN {X 0,Y 294.475,Z 361.687,A -85,B 0,C 180,E1 -16632.679,E2 -16632.679} C_VEL
LIN {X 0,Y 292.856,Z 370.762,A -85,B 0,C 180,E1 -16634.693,E2 -16634.693} C_VEL
LIN {X 0,Y 291.554,Z 378.206,A -85,B 0,C 180,E1 -16636.761,E2 -16636.761} C_VEL
LIN {X 0,Y 290.602,Z 384.189,A -85,B 0,C 180,E1 -16638.844,E2 -16638.844} C_VEL
LIN {X 0,Y 289.981,Z 388.922,A -85,B 0,C 180,E1 -16640.936,E2 -16640.936} C_VEL
LIN {X 0,Y 289.57,Z 392.539,A -85,B 0,C 180,E1 -16643.029,E2 -16643.029} C_VEL
LIN {X 0,Y 289.475,Z 394.504,A -85,B 0,C 180,E1 -16644.513,E2 -16644.513} C_VEL
LIN {X 0,Y 289.473,Z 396.814,A -85,B 0,C 180,E1 -16647.216,E2 -16647.216} C_VEL
LIN {X 0,Y 289.45,Z 397.423,A -85,B 0,C 180,E1 -16648.608,E2 -16648.608} C_VEL
LIN {X 0,Y 289.494,Z 397.639,A -85,B 0,C 180,E1 -16649.999,E2 -16649.999} C_VEL
LIN {X 0,Y 289.45,Z 397.415,A -85,B 0,C 180,E1 -16651.391,E2 -16651.391} C_VEL
LIN {X 0,Y 289.474,Z 396.802,A -85,B 0,C 180,E1 -16652.782,E2 -16652.782} C_VEL
LIN {X 0,Y 289.458,Z 394.519,A -85,B 0,C 180,E1 -16655.451,E2 -16655.451} C_VEL
LIN {X 0,Y 289.712,Z 391.428,A -85,B 0,C 180,E1 -16657.667,E2 -16657.667} C_VEL
LIN {X 0,Y 290.147,Z 387.431,A -85,B 0,C 180,E1 -16659.761,E2 -16659.761} C_VEL
LIN {X 0,Y 290.983,Z 381.291,A -85,B 0,C 180,E1 -16662.2,E2 -16662.2} C_VEL
LIN {X 0,Y 292.205,Z 374.597,A -85,B 0,C 180,E1 -16664.271,E2 -16664.271} C_VEL
LIN {X 0,Y 293.697,Z 366.295,A -85,B 0,C 180,E1 -16666.329,E2 -16666.329} C_VEL
LIN {X 0,Y 295.039,Z 357.779,A -85,B 0,C 180,E1 -16668.038,E2 -16668.038} C_VEL
LIN {X 0,Y 296.777,Z 347.268,A -85,B 0,C 180,E1 -16669.721,E2 -16669.721} C_VEL
LIN {X 0,Y 298.643,Z 335.443,A -85,B 0,C 180,E1 -16671.211,E2 -16671.211} C_VEL
LIN {X 0,Y 300.208,Z 323.536,A -85,B 0,C 180,E1 -16672.359,E2 -16672.359} C_VEL
LIN {X 0,Y 301.593,Z 311.148,A -85,B 0,C 180,E1 -16673.246,E2 -16673.246} C_VEL
LIN {X 0,Y 302.718,Z 298.399,A -85,B 0,C 180,E1 -16673.88,E2 -16673.88} C_VEL
LIN {X 0,Y 303.295,Z 284.93,A -85,B 0,C 180,E1 -16674.286,E2 -16674.286} C_VEL
LIN {X 0,Y 304.553,Z 229.213,A -85,B 0,C 180,E1 -16675.596,E2 -16675.596} C_VEL
LIN {X 0,Y 300.379,Z 202.018,A -85,B 0,C 180,E1 -16676.682,E2 -16676.682} C_VEL
LIN {X 0,Y 297.761,Z 188.813,A -85,B 0,C 180,E1 -16677.282,E2 -16677.282} C_VEL
LIN {X 0,Y 296.19,Z 184.396,A -85,B 0,C 180,E1 -16677.587,E2 -16677.587} C_VEL
LIN {X 0,Y 294.225,Z 174.62,A -85,B 0,C 180,E1 -16680.693,E2 -16680.693} C_VEL
LIN {X 0,Y 291.98,Z 164.696,A -85,B 0,C 180,E1 -16684.015,E2 -16684.015} C_VEL
LIN {X 0,Y 291.365,Z 162.187,A -85,B 0,C 180,E1 -16684.904,E2 -16684.904} C_VEL
LIN {X 0,Y 291.355,Z 162.182,A -85,B 0,C 180,E1 -16687.248,E2 -16687.248} C_VEL
LIN {X 0,Y 291.296,Z 162.197,A -85,B 0,C 180,E1 -16690.647,E2 -16690.647} C_VEL
LIN {X 0,Y 291.277,Z 162.201,A -85,B 0,C 180,E1 -16694.403,E2 -16694.403} C_VEL
LIN {X 0,Y 291.29,Z 162.2,A -85,B 0,C 180,E1 -16698.41,E2 -16698.41} C_VEL
LIN {X 0,Y 291.328,Z 162.198,A -85,B 0,C 180,E1 -16701.154,E2 -16701.154} C_VEL
LIN {X 0,Y 291.349,Z 162.193,A -85,B 0,C 180,E1 -16704.624,E2 -16704.624} C_VEL
LIN {X 0,Y 291.359,Z 162.187,A -85,B 0,C 180,E1 -16707.949,E2 -16707.949} C_VEL
LIN {X 0,Y 291.335,Z 162.188,A -85,B 0,C 180,E1 -16711.153,E2 -16711.153} C_VEL
LIN {X 0,Y 291.336,Z 162.193,A -85,B 0,C 180,E1 -16714.264,E2 -16714.264} C_VEL
LIN {X 0,Y 291.341,Z 162.187,A -85,B 0,C 180,E1 -16717.296,E2 -16717.296} C_VEL
LIN {X 0,Y 291.377,Z 162.19,A -85,B 0,C 180,E1 -16720.264,E2 -16720.264} C_VEL
LIN {X 0,Y 291.466,Z 162.177,A -85,B 0,C 180,E1 -16724.682,E2 -16724.682} C_VEL
LIN {X 0,Y 291.517,Z 162.167,A -85,B 0,C 180,E1 -16728.88,E2 -16728.88} C_VEL
LIN {X 0,Y 291.621,Z 162.154,A -85,B 0,C 180,E1 -16731.686,E2 -16731.686} C_VEL
LIN {X 0,Y 291.586,Z 162.163,A -85,B 0,C 180,E1 -16734.468,E2 -16734.468} C_VEL
LIN {X 0,Y 291.859,Z 162.125,A -85,B 0,C 180,E1 -16738.62,E2 -16738.62} C_VEL
LIN {X 0,Y 291.861,Z 162.128,A -85,B 0,C 180,E1 -16741.38,E2 -16741.38} C_VEL
LIN {X 0,Y 291.678,Z 162.148,A -85,B 0,C 180,E1 -16746.92,E2 -16746.92} C_VEL
LIN {X 0,Y 291.56,Z 162.168,A -85,B 0,C 180,E1 -16749.714,E2 -16749.714} C_VEL
LIN {X 0,Y 291.473,Z 162.176,A -85,B 0,C 180,E1 -16753.953,E2 -16753.953} C_VEL
LIN {X 0,Y 291.397,Z 162.186,A -85,B 0,C 180,E1 -16756.823,E2 -16756.823} C_VEL
LIN {X 0,Y 291.384,Z 162.184,A -85,B 0,C 180,E1 -16759.843,E2 -16759.843} C_VEL
LIN {X 0,Y 291.338,Z 162.191,A -85,B 0,C 180,E1 -16764.211,E2 -16764.211} C_VEL
LIN {X 0,Y 291.344,Z 162.192,A -85,B 0,C 180,E1 -16767.28,E2 -16767.28} C_VEL
LIN {X 0,Y 291.312,Z 162.195,A -85,B 0,C 180,E1 -16770.44,E2 -16770.44} C_VEL
LIN {X 0,Y 291.337,Z 162.193,A -85,B 0,C 180,E1 -16773.7,E2 -16773.7} C_VEL
LIN {X 0,Y 291.353,Z 162.192,A -85,B 0,C 180,E1 -16777.25,E2 -16777.25} C_VEL
LIN {X 0,Y 291.295,Z 162.2,A -85,B 0,C 180,E1 -16780.649,E2 -16780.649} C_VEL
LIN {X 0,Y 291.278,Z 162.202,A -85,B 0,C 180,E1 -16784.405,E2 -16784.405} C_VEL
LIN {X 0,Y 291.313,Z 162.196,A -85,B 0,C 180,E1 -16788.408,E2 -16788.408} C_VEL
LIN {X 0,Y 291.34,Z 162.191,A -85,B 0,C 180,E1 -16791.158,E2 -16791.158} C_VEL
LIN {X 0,Y 291.353,Z 162.193,A -85,B 0,C 180,E1 -16794.626,E2 -16794.626} C_VEL
LIN {X 0,Y 291.364,Z 162.193,A -85,B 0,C 180,E1 -16797.951,E2 -16797.951} C_VEL
LIN {X 0,Y 291.391,Z 162.221,A -85,B 0,C 180,E1 -16800.794,E2 -16800.794} C_VEL
LIN {X 0,Y 292.247,Z 165.894,A -85,B 0,C 180,E1 -16802.1,E2 -16802.1} C_VEL
LIN {X 0,Y 301.013,Z 185.995,A -85,B 0,C 180,E1 -16803.518,E2 -16803.518} C_VEL
LIN {X 0,Y 305.302,Z 197.565,A -85,B 0,C 180,E1 -16804.22,E2 -16804.22} C_VEL
LIN {X 0,Y 304.513,Z 233.459,A -85,B 0,C 180,E1 -16805.068,E2 -16805.068} C_VEL
LIN {X 0,Y 303.399,Z 273.689,A -85,B 0,C 180,E1 -16806.041,E2 -16806.041} C_VEL
LIN {X 0,Y 302.639,Z 287.422,A -85,B 0,C 180,E1 -16806.658,E2 -16806.658} C_VEL
LIN {X 0,Y 301.671,Z 298.652,A -85,B 0,C 180,E1 -16807.395,E2 -16807.395} C_VEL
LIN {X 0,Y 300.361,Z 309.973,A -85,B 0,C 180,E1 -16808.376,E2 -16808.376} C_VEL
LIN {X 0,Y 298.768,Z 321.607,A -85,B 0,C 180,E1 -16809.699,E2 -16809.699} C_VEL
LIN {X 0,Y 297.445,Z 331.502,A -85,B 0,C 180,E1 -16811.131,E2 -16811.131} C_VEL
LIN {X 0,Y 295.927,Z 340.571,A -85,B 0,C 180,E1 -16812.732,E2 -16812.732} C_VEL
LIN {X 0,Y 294.489,Z 348.428,A -85,B 0,C 180,E1 -16814.427,E2 -16814.427} C_VEL
LIN {X 0,Y 293.005,Z 356.105,A -85,B 0,C 180,E1 -16816.476,E2 -16816.476} C_VEL
LIN {X 0,Y 291.688,Z 363.147,A -85,B 0,C 180,E1 -16818.887,E2 -16818.887} C_VEL
LIN {X 0,Y 290.813,Z 367.837,A -85,B 0,C 180,E1 -16820.963,E2 -16820.963} C_VEL
LIN {X 0,Y 290.23,Z 371.555,A -85,B 0,C 180,E1 -16823.135,E2 -16823.135} C_VEL
LIN {X 0,Y 290.025,Z 373.271,A -85,B 0,C 180,E1 -16824.438,E2 -16824.438} C_VEL
LIN {X 0,Y 289.823,Z 374.664,A -85,B 0,C 180,E1 -16825.829,E2 -16825.829} C_VEL
LIN {X 0,Y 289.519,Z 376.266,A -85,B 0,C 180,E1 -16828.61,E2 -16828.61} C_VEL
LIN {X 0,Y 289.505,Z 376.496,A -85,B 0,C 180,E1 -16830.001,E2 -16830.001} C_VEL
LIN {X 0,Y 289.518,Z 376.305,A -85,B 0,C 180,E1 -16831.392,E2 -16831.392} C_VEL
LIN {X 0,Y 289.816,Z 374.753,A -85,B 0,C 180,E1 -16834.173,E2 -16834.173} C_VEL
LIN {X 0,Y 290.009,Z 373.399,A -85,B 0,C 180,E1 -16835.563,E2 -16835.563} C_VEL
LIN {X 0,Y 290.419,Z 370.539,A -85,B 0,C 180,E1 -16837.649,E2 -16837.649} C_VEL
LIN {X 0,Y 290.986,Z 366.662,A -85,B 0,C 180,E1 -16839.734,E2 -16839.734} C_VEL
LIN {X 0,Y 292.01,Z 361.648,A -85,B 0,C 180,E1 -16841.805,E2 -16841.805} C_VEL
LIN {X 0,Y 293.194,Z 355.338,A -85,B 0,C 180,E1 -16843.87,E2 -16843.87} C_VEL
LIN {X 0,Y 294.656,Z 347.438,A -85,B 0,C 180,E1 -16845.92,E2 -16845.92} C_VEL
LIN {X 0,Y 296.498,Z 337.605,A -85,B 0,C 180,E1 -16847.948,E2 -16847.948} C_VEL
LIN {X 0,Y 298.054,Z 327.285,A -85,B 0,C 180,E1 -16849.634,E2 -16849.634} C_VEL
LIN {X 0,Y 299.551,Z 317.056,A -85,B 0,C 180,E1 -16850.965,E2 -16850.965} C_VEL
LIN {X 0,Y 300.986,Z 305.859,A -85,B 0,C 180,E1 -16852.119,E2 -16852.119} C_VEL
LIN {X 0,Y 302.211,Z 293.229,A -85,B 0,C 180,E1 -16853.106,E2 -16853.106} C_VEL
LIN {X 0,Y 303.128,Z 280.557,A -85,B 0,C 180,E1 -16853.801,E2 -16853.801} C_VEL
LIN {X 0,Y 303.825,Z 267.49,A -85,B 0,C 180,E1 -16854.242,E2 -16854.242} C_VEL
LIN {X 0,Y 305.427,Z 198.024,A -85,B 0,C 180,E1 -16855.876,E2 -16855.876} C_VEL
LIN {X 0,Y 301.019,Z 185.907,A -85,B 0,C 180,E1 -16856.605,E2 -16856.605} C_VEL
LIN {X 0,Y 293.507,Z 168.701,A -85,B 0,C 180,E1 -16857.816,E2 -16857.816} C_VEL
LIN {X 0,Y 292.229,Z 165.692,A -85,B 0,C 180,E1 -16858.074,E2 -16858.074} C_VEL
LIN {X 0,Y 291.367,Z 162.192,A -85,B 0,C 180,E1 -16859.432,E2 -16859.432} C_VEL
LIN {X 0,Y 291.341,Z 162.192,A -85,B 0,C 180,E1 -16862.402,E2 -16862.402} C_VEL
LIN {X 0,Y 291.357,Z 162.193,A -85,B 0,C 180,E1 -16865.375,E2 -16865.375} C_VEL
LIN {X 0,Y 291.31,Z 162.197,A -85,B 0,C 180,E1 -16868.849,E2 -16868.849} C_VEL
LIN {X 0,Y 291.289,Z 162.199,A -85,B 0,C 180,E1 -16872.498,E2 -16872.498} C_VEL
LIN {X 0,Y 291.29,Z 162.196,A -85,B 0,C 180,E1 -16876.37,E2 -16876.37} C_VEL
LIN {X 0,Y 291.356,Z 162.186,A -85,B 0,C 180,E1 -16880.524,E2 -16880.524} C_VEL
LIN {X 0,Y 291.39,Z 162.189,A -85,B 0,C 180,E1 -16882.917,E2 -16882.917} C_VEL
LIN {X 0,Y 291.346,Z 162.187,A -85,B 0,C 180,E1 -16885.491,E2 -16885.491} C_VEL
LIN {X 0,Y 290.652,Z 162.278,A -85,B 0,C 180,E1 -16886.645,E2 -16886.645} C_VEL
LIN {X 0,Y 287.787,Z 162.636,A -85,B 0,C 180,E1 -16888.523,E2 -16888.523} C_VEL
LIN {X 0,Y 285.377,Z 162.931,A -85,B 0,C 180,E1 -16890.049,E2 -16890.049} C_VEL
LIN {X 0,Y 284.354,Z 163.059,A -85,B 0,C 180,E1 -16891.23,E2 -16891.23} C_VEL
LIN {X 0,Y 284.276,Z 163.066,A -85,B 0,C 180,E1 -16891.631,E2 -16891.631} C_VEL
LIN {X 0,Y 284.309,Z 163.068,A -85,B 0,C 180,E1 -16895.15,E2 -16895.15} C_VEL
LIN {X 0,Y 284.315,Z 163.06,A -85,B 0,C 180,E1 -16898.236,E2 -16898.236} C_VEL
LIN {X 0,Y 284.33,Z 163.066,A -85,B 0,C 180,E1 -16901.256,E2 -16901.256} C_VEL
LIN {X 0,Y 284.418,Z 163.046,A -85,B 0,C 180,E1 -16905.694,E2 -16905.694} C_VEL
LIN {X 0,Y 284.513,Z 163.045,A -85,B 0,C 180,E1 -16910.043,E2 -16910.043} C_VEL
LIN {X 0,Y 284.639,Z 163.017,A -85,B 0,C 180,E1 -16912.908,E2 -16912.908} C_VEL
LIN {X 0,Y 284.835,Z 163.001,A -85,B 0,C 180,E1 -16918.586,E2 -16918.586} C_VEL
LIN {X 0,Y 284.834,Z 162.992,A -85,B 0,C 180,E1 -16921.414,E2 -16921.414} C_VEL
LIN {X 0,Y 284.635,Z 163.026,A -85,B 0,C 180,E1 -16927.092,E2 -16927.092} C_VEL
LIN {X 0,Y 284.508,Z 163.037,A -85,B 0,C 180,E1 -16929.957,E2 -16929.957} C_VEL
LIN {X 0,Y 284.404,Z 163.055,A -85,B 0,C 180,E1 -16934.307,E2 -16934.307} C_VEL
LIN {X 0,Y 284.328,Z 163.058,A -85,B 0,C 180,E1 -16937.254,E2 -16937.254} C_VEL
LIN {X 0,Y 284.321,Z 163.067,A -85,B 0,C 180,E1 -16940.247,E2 -16940.247} C_VEL
LIN {X 0,Y 284.292,Z 163.068,A -85,B 0,C 180,E1 -16943.84,E2 -16943.84} C_VEL
LIN {X 0,Y 284.279,Z 163.069,A -85,B 0,C 180,E1 -16948.016,E2 -16948.016} C_VEL
LIN {X 0,Y 284.284,Z 163.075,A -85,B 0,C 180,E1 -16951.276,E2 -16951.276} C_VEL
LIN {X 0,Y 284.336,Z 163.068,A -85,B 0,C 180,E1 -16955.346,E2 -16955.346} C_VEL
LIN {X 0,Y 284.297,Z 163.066,A -85,B 0,C 180,E1 -16958.171,E2 -16958.171} C_VEL
LIN {X 0,Y 284.237,Z 163.076,A -85,B 0,C 180,E1 -16962.117,E2 -16962.117} C_VEL
LIN {X 0,Y 284.237,Z 163.078,A -85,B 0,C 180,E1 -16966.186,E2 -16966.186} C_VEL
LIN {X 0,Y 284.284,Z 163.07,A -85,B 0,C 180,E1 -16970.03,E2 -16970.03} C_VEL
LIN {X 0,Y 284.312,Z 163.072,A -85,B 0,C 180,E1 -16974.199,E2 -16974.199} C_VEL
LIN {X 0,Y 284.323,Z 163.144,A -85,B 0,C 180,E1 -16974.492,E2 -16974.492} C_VEL
LIN {X 0,Y 286.57,Z 172.422,A -85,B 0,C 180,E1 -16977.764,E2 -16977.764} C_VEL
LIN {X 0,Y 288.945,Z 183.883,A -85,B 0,C 180,E1 -16981.561,E2 -16981.561} C_VEL
LIN {X 0,Y 289.148,Z 184.766,A -85,B 0,C 180,E1 -16981.698,E2 -16981.698} C_VEL
LIN {X 0,Y 292.301,Z 193.296,A -85,B 0,C 180,E1 -16982.259,E2 -16982.259} C_VEL
LIN {X 0,Y 296.789,Z 220.039,A -85,B 0,C 180,E1 -16983.418,E2 -16983.418} C_VEL
LIN {X 0,Y 298.232,Z 230.245,A -85,B 0,C 180,E1 -16983.824,E2 -16983.824} C_VEL
LIN {X 0,Y 296.587,Z 293.213,A -85,B 0,C 180,E1 -16985.36,E2 -16985.36} C_VEL
LIN {X 0,Y 295.566,Z 307.137,A -85,B 0,C 180,E1 -16985.971,E2 -16985.971} C_VEL
LIN {X 0,Y 294.182,Z 319.59,A -85,B 0,C 180,E1 -16986.784,E2 -16986.784} C_VEL
LIN {X 0,Y 292.706,Z 330.7,A -85,B 0,C 180,E1 -16987.78,E2 -16987.78} C_VEL
LIN {X 0,Y 290.959,Z 342.282,A -85,B 0,C 180,E1 -16989.128,E2 -16989.128} C_VEL
LIN {X 0,Y 289.132,Z 352.712,A -85,B 0,C 180,E1 -16990.659,E2 -16990.659} C_VEL
LIN {X 0,Y 287.521,Z 362.231,A -85,B 0,C 180,E1 -16992.42,E2 -16992.42} C_VEL
LIN {X 0,Y 285.979,Z 370.504,A -85,B 0,C 180,E1 -16994.316,E2 -16994.316} C_VEL
LIN {X 0,Y 284.631,Z 377.948,A -85,B 0,C 180,E1 -16996.433,E2 -16996.433} C_VEL
LIN {X 0,Y 283.577,Z 383.929,A -85,B 0,C 180,E1 -16998.564,E2 -16998.564} C_VEL
LIN {X 0,Y 282.933,Z 388.662,A -85,B 0,C 180,E1 -17000.708,E2 -17000.708} C_VEL
LIN {X 0,Y 282.496,Z 392.28,A -85,B 0,C 180,E1 -17002.854,E2 -17002.854} C_VEL
LIN {X 0,Y 282.37,Z 394.486,A -85,B 0,C 180,E1 -17004.609,E2 -17004.609} C_VEL
LIN {X 0,Y 282.377,Z 396.554,A -85,B 0,C 180,E1 -17007.146,E2 -17007.146} C_VEL
LIN {X 0,Y 282.372,Z 397.165,A -85,B 0,C 180,E1 -17008.573,E2 -17008.573} C_VEL
LIN {X 0,Y 282.411,Z 397.38,A -85,B 0,C 180,E1 -17009.999,E2 -17009.999} C_VEL
LIN {X 0,Y 282.372,Z 397.157,A -85,B 0,C 180,E1 -17011.425,E2 -17011.425} C_VEL
LIN {X 0,Y 282.377,Z 396.542,A -85,B 0,C 180,E1 -17012.852,E2 -17012.852} C_VEL
LIN {X 0,Y 282.372,Z 394.456,A -85,B 0,C 180,E1 -17015.395,E2 -17015.395} C_VEL
LIN {X 0,Y 282.666,Z 391.167,A -85,B 0,C 180,E1 -17017.859,E2 -17017.859} C_VEL
LIN {X 0,Y 283.121,Z 387.17,A -85,B 0,C 180,E1 -17020.006,E2 -17020.006} C_VEL
LIN {X 0,Y 284.019,Z 381.029,A -85,B 0,C 180,E1 -17022.504,E2 -17022.504} C_VEL
LIN {X 0,Y 285.315,Z 374.335,A -85,B 0,C 180,E1 -17024.623,E2 -17024.623} C_VEL
LIN {X 0,Y 286.853,Z 366.032,A -85,B 0,C 180,E1 -17026.73,E2 -17026.73} C_VEL
LIN {X 0,Y 288.27,Z 357.516,A -85,B 0,C 180,E1 -17028.477,E2 -17028.477} C_VEL
LIN {X 0,Y 290.087,Z 347.004,A -85,B 0,C 180,E1 -17030.195,E2 -17030.195} C_VEL
LIN {X 0,Y 292.024,Z 335.179,A -85,B 0,C 180,E1 -17031.716,E2 -17031.716} C_VEL
LIN {X 0,Y 293.662,Z 323.271,A -85,B 0,C 180,E1 -17032.885,E2 -17032.885} C_VEL
LIN {X 0,Y 295.1,Z 310.881,A -85,B 0,C 180,E1 -17033.788,E2 -17033.788} C_VEL
LIN {X 0,Y 296.229,Z 298.128,A -85,B 0,C 180,E1 -17034.436,E2 -17034.436} C_VEL
LIN {X 0,Y 296.828,Z 284.649,A -85,B 0,C 180,E1 -17034.85,E2 -17034.85} C_VEL
LIN {X 0,Y 298.068,Z 229.709,A -85,B 0,C 180,E1 -17036.174,E2 -17036.174} C_VEL
LIN {X 0,Y 294.324,Z 204.887,A -85,B 0,C 180,E1 -17037.192,E2 -17037.192} C_VEL
LIN {X 0,Y 291.7,Z 191.207,A -85,B 0,C 180,E1 -17037.825,E2 -17037.825} C_VEL
LIN {X 0,Y 288.986,Z 184.174,A -85,B 0,C 180,E1 -17038.313,E2 -17038.313} C_VEL
LIN {X 0,Y 286.763,Z 173.628,A -85,B 0,C 180,E1 -17041.796,E2 -17041.796} C_VEL
LIN {X 0,Y 284.688,Z 164.568,A -85,B 0,C 180,E1 -17044.952,E2 -17044.952} C_VEL
LIN {X 0,Y 284.309,Z 163.067,A -85,B 0,C 180,E1 -17045.582,E2 -17045.582} C_VEL
LIN {X 0,Y 284.294,Z 163.067,A -85,B 0,C 180,E1 -17048.17,E2 -17048.17} C_VEL
LIN {X 0,Y 284.233,Z 163.077,A -85,B 0,C 180,E1 -17052.116,E2 -17052.116} C_VEL
LIN {X 0,Y 284.232,Z 163.078,A -85,B 0,C 180,E1 -17056.185,E2 -17056.185} C_VEL
LIN {X 0,Y 284.278,Z 163.071,A -85,B 0,C 180,E1 -17060.029,E2 -17060.029} C_VEL
LIN {X 0,Y 284.315,Z 163.067,A -85,B 0,C 180,E1 -17063.611,E2 -17063.611} C_VEL
LIN {X 0,Y 284.3,Z 163.067,A -85,B 0,C 180,E1 -17067.19,E2 -17067.19} C_VEL
LIN {X 0,Y 284.33,Z 163.066,A -85,B 0,C 180,E1 -17070.373,E2 -17070.373} C_VEL
LIN {X 0,Y 284.29,Z 163.069,A -85,B 0,C 180,E1 -17073.578,E2 -17073.578} C_VEL
LIN {X 0,Y 284.3,Z 163.065,A -85,B 0,C 180,E1 -17076.701,E2 -17076.701} C_VEL
LIN {X 0,Y 284.326,Z 163.066,A -85,B 0,C 180,E1 -17079.928,E2 -17079.928} C_VEL
LIN {X 0,Y 284.407,Z 163.054,A -85,B 0,C 180,E1 -17084.516,E2 -17084.516} C_VEL
LIN {X 0,Y 284.449,Z 163.048,A -85,B 0,C 180,E1 -17088.6,E2 -17088.6} C_VEL
LIN {X 0,Y 284.572,Z 163.031,A -85,B 0,C 180,E1 -17091.479,E2 -17091.479} C_VEL
LIN {X 0,Y 284.556,Z 163.039,A -85,B 0,C 180,E1 -17094.33,E2 -17094.33} C_VEL
LIN {X 0,Y 284.827,Z 163.001,A -85,B 0,C 180,E1 -17098.586,E2 -17098.586} C_VEL
LIN {X 0,Y 284.828,Z 163.005,A -85,B 0,C 180,E1 -17101.414,E2 -17101.414} C_VEL
LIN {X 0,Y 284.634,Z 163.025,A -85,B 0,C 180,E1 -17107.092,E2 -17107.092} C_VEL
LIN {X 0,Y 284.506,Z 163.044,A -85,B 0,C 180,E1 -17109.958,E2 -17109.958} C_VEL
LIN {X 0,Y 284.41,Z 163.054,A -85,B 0,C 180,E1 -17114.307,E2 -17114.307} C_VEL
LIN {X 0,Y 284.316,Z 163.064,A -85,B 0,C 180,E1 -17118.745,E2 -17118.745} C_VEL
LIN {X 0,Y 284.319,Z 163.071,A -85,B 0,C 180,E1 -17123.297,E2 -17123.297} C_VEL
LIN {X 0,Y 284.319,Z 163.065,A -85,B 0,C 180,E1 -17127.146,E2 -17127.146} C_VEL
LIN {X 0,Y 284.29,Z 163.07,A -85,B 0,C 180,E1 -17130.092,E2 -17130.092} C_VEL
LIN {X 0,Y 284.298,Z 163.069,A -85,B 0,C 180,E1 -17132.946,E2 -17132.946} C_VEL
LIN {X 0,Y 284.315,Z 163.068,A -85,B 0,C 180,E1 -17136.389,E2 -17136.389} C_VEL
LIN {X 0,Y 284.277,Z 163.072,A -85,B 0,C 180,E1 -17140,E2 -17140} C_VEL
LIN {X 0,Y 284.229,Z 163.079,A -85,B 0,C 180,E1 -17144.189,E2 -17144.189} C_VEL
LIN {X 0,Y 284.254,Z 163.076,A -85,B 0,C 180,E1 -17148.123,E2 -17148.123} C_VEL
LIN {X 0,Y 284.299,Z 163.068,A -85,B 0,C 180,E1 -17151.831,E2 -17151.831} C_VEL
LIN {X 0,Y 284.304,Z 163.071,A -85,B 0,C 180,E1 -17155.352,E2 -17155.352} C_VEL
LIN {X 0,Y 284.283,Z 163.073,A -85,B 0,C 180,E1 -17158.726,E2 -17158.726} C_VEL
LIN {X 0,Y 284.341,Z 163.119,A -85,B 0,C 180,E1 -17160.21,E2 -17160.21} C_VEL
LIN {X 0,Y 285.068,Z 166.127,A -85,B 0,C 180,E1 -17161.331,E2 -17161.331} C_VEL
LIN {X 0,Y 294.427,Z 187.245,A -85,B 0,C 180,E1 -17162.903,E2 -17162.903} C_VEL
LIN {X 0,Y 299.04,Z 199.561,A -85,B 0,C 180,E1 -17163.685,E2 -17163.685} C_VEL
LIN {X 0,Y 297.076,Z 271.387,A -85,B 0,C 180,E1 -17165.405,E2 -17165.405} C_VEL
LIN {X 0,Y 296.398,Z 283.881,A -85,B 0,C 180,E1 -17165.904,E2 -17165.904} C_VEL
LIN {X 0,Y 295.335,Z 296.665,A -85,B 0,C 180,E1 -17166.697,E2 -17166.697} C_VEL
LIN {X 0,Y 294.022,Z 308.501,A -85,B 0,C 180,E1 -17167.701,E2 -17167.701} C_VEL
LIN {X 0,Y 292.542,Z 319.24,A -85,B 0,C 180,E1 -17168.879,E2 -17168.879} C_VEL
LIN {X 0,Y 291.109,Z 329.106,A -85,B 0,C 180,E1 -17170.247,E2 -17170.247} C_VEL
LIN {X 0,Y 289.541,Z 339.058,A -85,B 0,C 180,E1 -17171.973,E2 -17171.973} C_VEL
LIN {X 0,Y 287.899,Z 347.214,A -85,B 0,C 180,E1 -17173.697,E2 -17173.697} C_VEL
LIN {X 0,Y 286.361,Z 355.198,A -85,B 0,C 180,E1 -17175.794,E2 -17175.794} C_VEL
LIN {X 0,Y 285.113,Z 361.602,A -85,B 0,C 180,E1 -17177.906,E2 -17177.906} C_VEL
LIN {X 0,Y 284.049,Z 366.684,A -85,B 0,C 180,E1 -17180.027,E2 -17180.027} C_VEL
LIN {X 0,Y 283.366,Z 370.624,A -85,B 0,C 180,E1 -17182.161,E2 -17182.161} C_VEL
LIN {X 0,Y 282.967,Z 373.531,A -85,B 0,C 180,E1 -17184.299,E2 -17184.299} C_VEL
LIN {X 0,Y 282.767,Z 374.922,A -85,B 0,C 180,E1 -17185.725,E2 -17185.725} C_VEL
LIN {X 0,Y 282.44,Z 376.525,A -85,B 0,C 180,E1 -17188.575,E2 -17188.575} C_VEL
LIN {X 0,Y 282.423,Z 376.755,A -85,B 0,C 180,E1 -17190.001,E2 -17190.001} C_VEL
LIN {X 0,Y 282.439,Z 376.564,A -85,B 0,C 180,E1 -17191.427,E2 -17191.427} C_VEL
LIN {X 0,Y 282.76,Z 375.011,A -85,B 0,C 180,E1 -17194.277,E2 -17194.277} C_VEL
LIN {X 0,Y 283.205,Z 372.105,A -85,B 0,C 180,E1 -17196.954,E2 -17196.954} C_VEL
LIN {X 0,Y 283.754,Z 368.33,A -85,B 0,C 180,E1 -17199.265,E2 -17199.265} C_VEL
LIN {X 0,Y 284.661,Z 363.704,A -85,B 0,C 180,E1 -17201.392,E2 -17201.392} C_VEL
LIN {X 0,Y 286.076,Z 356.726,A -85,B 0,C 180,E1 -17203.859,E2 -17203.859} C_VEL
LIN {X 0,Y 287.556,Z 349.162,A -85,B 0,C 180,E1 -17205.96,E2 -17205.96} C_VEL
LIN {X 0,Y 289.437,Z 339.634,A -85,B 0,C 180,E1 -17208.035,E2 -17208.035} C_VEL
LIN {X 0,Y 291.072,Z 329.802,A -85,B 0,C 180,E1 -17209.758,E2 -17209.758} C_VEL
LIN {X 0,Y 292.535,Z 320.122,A -85,B 0,C 180,E1 -17211.123,E2 -17211.123} C_VEL
LIN {X 0,Y 293.933,Z 309.634,A -85,B 0,C 180,E1 -17212.308,E2 -17212.308} C_VEL
LIN {X 0,Y 295.409,Z 296.996,A -85,B 0,C 180,E1 -17213.392,E2 -17213.392} C_VEL
LIN {X 0,Y 296.416,Z 284.334,A -85,B 0,C 180,E1 -17214.189,E2 -17214.189} C_VEL
LIN {X 0,Y 297.186,Z 272.235,A -85,B 0,C 180,E1 -17214.68,E2 -17214.68} C_VEL
LIN {X 0,Y 299.125,Z 199.604,A -85,B 0,C 180,E1 -17216.428,E2 -17216.428} C_VEL
LIN {X 0,Y 292.94,Z 183.604,A -85,B 0,C 180,E1 -17217.47,E2 -17217.47} C_VEL
LIN {X 0,Y 285.051,Z 166.049,A -85,B 0,C 180,E1 -17218.822,E2 -17218.822} C_VEL
LIN {X 0,Y 284.325,Z 163.071,A -85,B 0,C 180,E1 -17219.96,E2 -17219.96} C_VEL
LIN {X 0,Y 284.306,Z 163.07,A -85,B 0,C 180,E1 -17222.945,E2 -17222.945} C_VEL
LIN {X 0,Y 284.321,Z 163.066,A -85,B 0,C 180,E1 -17226.388,E2 -17226.388} C_VEL
LIN {X 0,Y 284.256,Z 163.077,A -85,B 0,C 180,E1 -17230.003,E2 -17230.003} C_VEL
LIN {X 0,Y 284.235,Z 163.078,A -85,B 0,C 180,E1 -17234.188,E2 -17234.188} C_VEL
LIN {X 0,Y 284.241,Z 163.076,A -85,B 0,C 180,E1 -17238.118,E2 -17238.118} C_VEL
LIN {X 0,Y 284.309,Z 163.068,A -85,B 0,C 180,E1 -17242.282,E2 -17242.282} C_VEL
LIN {X 0,Y 284.299,Z 163.066,A -85,B 0,C 180,E1 -17245.473,E2 -17245.473} C_VEL
LIN {X 0,Y 284.285,Z 163.074,A -85,B 0,C 180,E1 -17248.724,E2 -17248.724} C_VEL
LIN {X 0,Y 284.276,Z 163.066,A -85,B 0,C 180,E1 -17251.631,E2 -17251.631} C_VEL
LIN {X 0,Y 283.627,Z 163.154,A -85,B 0,C 180,E1 -17252.814,E2 -17252.814} C_VEL
LIN {X 0,Y 280.804,Z 163.508,A -85,B 0,C 180,E1 -17254.742,E2 -17254.742} C_VEL
LIN {X 0,Y 278.393,Z 163.803,A -85,B 0,C 180,E1 -17256.307,E2 -17256.307} C_VEL
LIN {X 0,Y 277.346,Z 163.926,A -85,B 0,C 180,E1 -17257.52,E2 -17257.52} C_VEL
LIN {X 0,Y 277.254,Z 163.937,A -85,B 0,C 180,E1 -17257.931,E2 -17257.931} C_VEL
LIN {X 0,Y 277.298,Z 163.945,A -85,B 0,C 180,E1 -17260.763,E2 -17260.763} C_VEL
LIN {X 0,Y 277.37,Z 163.923,A -85,B 0,C 180,E1 -17265.322,E2 -17265.322} C_VEL
LIN {X 0,Y 277.456,Z 163.923,A -85,B 0,C 180,E1 -17269.787,E2 -17269.787} C_VEL
LIN {X 0,Y 277.598,Z 163.893,A -85,B 0,C 180,E1 -17272.728,E2 -17272.728} C_VEL
LIN {X 0,Y 277.802,Z 163.877,A -85,B 0,C 180,E1 -17278.55,E2 -17278.55} C_VEL
LIN {X 0,Y 277.801,Z 163.867,A -85,B 0,C 180,E1 -17281.45,E2 -17281.45} C_VEL
LIN {X 0,Y 277.59,Z 163.904,A -85,B 0,C 180,E1 -17287.273,E2 -17287.273} C_VEL
LIN {X 0,Y 277.449,Z 163.917,A -85,B 0,C 180,E1 -17290.213,E2 -17290.213} C_VEL
LIN {X 0,Y 277.363,Z 163.931,A -85,B 0,C 180,E1 -17294.678,E2 -17294.678} C_VEL
LIN {X 0,Y 277.267,Z 163.945,A -85,B 0,C 180,E1 -17299.239,E2 -17299.239} C_VEL
LIN {X 0,Y 277.245,Z 163.943,A -85,B 0,C 180,E1 -17302.349,E2 -17302.349} C_VEL
LIN {X 0,Y 277.231,Z 163.954,A -85,B 0,C 180,E1 -17305.529,E2 -17305.529} C_VEL
LIN {X 0,Y 277.237,Z 163.946,A -85,B 0,C 180,E1 -17308.793,E2 -17308.793} C_VEL
LIN {X 0,Y 277.239,Z 163.949,A -85,B 0,C 180,E1 -17312.164,E2 -17312.164} C_VEL
LIN {X 0,Y 277.273,Z 163.945,A -85,B 0,C 180,E1 -17315.796,E2 -17315.796} C_VEL
LIN {X 0,Y 277.216,Z 163.955,A -85,B 0,C 180,E1 -17319.331,E2 -17319.331} C_VEL
LIN {X 0,Y 277.191,Z 163.957,A -85,B 0,C 180,E1 -17323.202,E2 -17323.202} C_VEL
LIN {X 0,Y 277.192,Z 163.954,A -85,B 0,C 180,E1 -17327.33,E2 -17327.33} C_VEL
LIN {X 0,Y 277.253,Z 163.947,A -85,B 0,C 180,E1 -17331.796,E2 -17331.796} C_VEL
LIN {X 0,Y 277.307,Z 164.121,A -85,B 0,C 180,E1 -17333.889,E2 -17333.889} C_VEL
LIN {X 0,Y 279.864,Z 174.762,A -85,B 0,C 180,E1 -17337.748,E2 -17337.748} C_VEL
LIN {X 0,Y 281.839,Z 184.186,A -85,B 0,C 180,E1 -17340.886,E2 -17340.886} C_VEL
LIN {X 0,Y 286.203,Z 195.552,A -85,B 0,C 180,E1 -17341.684,E2 -17341.684} C_VEL
LIN {X 0,Y 290.498,Z 221.443,A -85,B 0,C 180,E1 -17342.841,E2 -17342.841} C_VEL
LIN {X 0,Y 291.868,Z 232.214,A -85,B 0,C 180,E1 -17343.268,E2 -17343.268} C_VEL
LIN {X 0,Y 290.139,Z 292.967,A -85,B 0,C 180,E1 -17344.775,E2 -17344.775} C_VEL
LIN {X 0,Y 289.18,Z 306.124,A -85,B 0,C 180,E1 -17345.357,E2 -17345.357} C_VEL
LIN {X 0,Y 287.807,Z 318.224,A -85,B 0,C 180,E1 -17346.143,E2 -17346.143} C_VEL
LIN {X 0,Y 286.149,Z 330.446,A -85,B 0,C 180,E1 -17347.242,E2 -17347.242} C_VEL
LIN {X 0,Y 284.314,Z 342.025,A -85,B 0,C 180,E1 -17348.616,E2 -17348.616} C_VEL
LIN {X 0,Y 282.395,Z 352.454,A -85,B 0,C 180,E1 -17350.178,E2 -17350.178} C_VEL
LIN {X 0,Y 280.893,Z 360.994,A -85,B 0,C 180,E1 -17351.775,E2 -17351.775} C_VEL
LIN {X 0,Y 279.438,Z 368.869,A -85,B 0,C 180,E1 -17353.564,E2 -17353.564} C_VEL
LIN {X 0,Y 277.911,Z 376.565,A -85,B 0,C 180,E1 -17355.725,E2 -17355.725} C_VEL
LIN {X 0,Y 276.566,Z 383.669,A -85,B 0,C 180,E1 -17358.27,E2 -17358.27} C_VEL
LIN {X 0,Y 275.904,Z 388.403,A -85,B 0,C 180,E1 -17360.469,E2 -17360.469} C_VEL
LIN {X 0,Y 275.448,Z 392.021,A -85,B 0,C 180,E1 -17362.67,E2 -17362.67} C_VEL
LIN {X 0,Y 275.263,Z 394.471,A -85,B 0,C 180,E1 -17364.714,E2 -17364.714} C_VEL
LIN {X 0,Y 275.283,Z 396.295,A -85,B 0,C 180,E1 -17367.072,E2 -17367.072} C_VEL
LIN {X 0,Y 275.295,Z 396.907,A -85,B 0,C 180,E1 -17368.536,E2 -17368.536} C_VEL
LIN {X 0,Y 275.33,Z 397.122,A -85,B 0,C 180,E1 -17369.999,E2 -17369.999} C_VEL
LIN {X 0,Y 275.295,Z 396.898,A -85,B 0,C 180,E1 -17371.462,E2 -17371.462} C_VEL
LIN {X 0,Y 275.284,Z 396.282,A -85,B 0,C 180,E1 -17372.926,E2 -17372.926} C_VEL
LIN {X 0,Y 275.283,Z 394.402,A -85,B 0,C 180,E1 -17375.33,E2 -17375.33} C_VEL
LIN {X 0,Y 275.592,Z 390.906,A -85,B 0,C 180,E1 -17378.062,E2 -17378.062} C_VEL
LIN {X 0,Y 276.111,Z 386.908,A -85,B 0,C 180,E1 -17380.263,E2 -17380.263} C_VEL
LIN {X 0,Y 277.04,Z 380.766,A -85,B 0,C 180,E1 -17382.824,E2 -17382.824} C_VEL
LIN {X 0,Y 278.431,Z 374.073,A -85,B 0,C 180,E1 -17384.993,E2 -17384.993} C_VEL
LIN {X 0,Y 280.027,Z 365.769,A -85,B 0,C 180,E1 -17387.15,E2 -17387.15} C_VEL
LIN {X 0,Y 281.509,Z 357.252,A -85,B 0,C 180,E1 -17388.937,E2 -17388.937} C_VEL
LIN {X 0,Y 283.435,Z 346.742,A -85,B 0,C 180,E1 -17390.691,E2 -17390.691} C_VEL
LIN {X 0,Y 285.426,Z 334.915,A -85,B 0,C 180,E1 -17392.244,E2 -17392.244} C_VEL
LIN {X 0,Y 287.129,Z 323.006,A -85,B 0,C 180,E1 -17393.436,E2 -17393.436} C_VEL
LIN {X 0,Y 288.63,Z 310.615,A -85,B 0,C 180,E1 -17394.356,E2 -17394.356} C_VEL
LIN {X 0,Y 289.787,Z 297.857,A -85,B 0,C 180,E1 -17395.017,E2 -17395.017} C_VEL
LIN {X 0,Y 290.405,Z 284.369,A -85,B 0,C 180,E1 -17395.439,E2 -17395.439} C_VEL
LIN {X 0,Y 291.711,Z 230.628,A -85,B 0,C 180,E1 -17396.757,E2 -17396.757} C_VEL
LIN {X 0,Y 287.813,Z 204.645,A -85,B 0,C 180,E1 -17397.859,E2 -17397.859} C_VEL
LIN {X 0,Y 285.715,Z 193.96,A -85,B 0,C 180,E1 -17398.376,E2 -17398.376} C_VEL
LIN {X 0,Y 281.729,Z 183.824,A -85,B 0,C 180,E1 -17399.126,E2 -17399.126} C_VEL
LIN {X 0,Y 279.492,Z 173.319,A -85,B 0,C 180,E1 -17402.725,E2 -17402.725} C_VEL
LIN {X 0,Y 277.272,Z 163.938,A -85,B 0,C 180,E1 -17406.17,E2 -17406.17} C_VEL
LIN {X 0,Y 277.212,Z 163.95,A -85,B 0,C 180,E1 -17409.33,E2 -17409.33} C_VEL
LIN {X 0,Y 277.187,Z 163.958,A -85,B 0,C 180,E1 -17413.201,E2 -17413.201} C_VEL
LIN {X 0,Y 277.187,Z 163.958,A -85,B 0,C 180,E1 -17417.329,E2 -17417.329} C_VEL
LIN {X 0,Y 277.246,Z 163.948,A -85,B 0,C 180,E1 -17421.795,E2 -17421.795} C_VEL
LIN {X 0,Y 277.271,Z 163.944,A -85,B 0,C 180,E1 -17424.339,E2 -17424.339} C_VEL
LIN {X 0,Y 277.233,Z 163.946,A -85,B 0,C 180,E1 -17427.835,E2 -17427.835} C_VEL
LIN {X 0,Y 277.231,Z 163.943,A -85,B 0,C 180,E1 -17431.206,E2 -17431.206} C_VEL
LIN {X 0,Y 277.225,Z 163.952,A -85,B 0,C 180,E1 -17434.471,E2 -17434.471} C_VEL
LIN {X 0,Y 277.239,Z 163.942,A -85,B 0,C 180,E1 -17437.651,E2 -17437.651} C_VEL
LIN {X 0,Y 277.269,Z 163.947,A -85,B 0,C 180,E1 -17440.761,E2 -17440.761} C_VEL
LIN {X 0,Y 277.363,Z 163.932,A -85,B 0,C 180,E1 -17445.322,E2 -17445.322} C_VEL
LIN {X 0,Y 277.443,Z 163.918,A -85,B 0,C 180,E1 -17449.786,E2 -17449.786} C_VEL
LIN {X 0,Y 277.583,Z 163.907,A -85,B 0,C 180,E1 -17452.727,E2 -17452.727} C_VEL
LIN {X 0,Y 277.794,Z 163.877,A -85,B 0,C 180,E1 -17458.55,E2 -17458.55} C_VEL
LIN {X 0,Y 277.795,Z 163.881,A -85,B 0,C 180,E1 -17461.45,E2 -17461.45} C_VEL
LIN {X 0,Y 277.592,Z 163.903,A -85,B 0,C 180,E1 -17467.273,E2 -17467.273} C_VEL
LIN {X 0,Y 277.446,Z 163.922,A -85,B 0,C 180,E1 -17470.214,E2 -17470.214} C_VEL
LIN {X 0,Y 277.363,Z 163.932,A -85,B 0,C 180,E1 -17474.678,E2 -17474.678} C_VEL
LIN {X 0,Y 277.273,Z 163.939,A -85,B 0,C 180,E1 -17479.239,E2 -17479.239} C_VEL
LIN {X 0,Y 277.266,Z 163.945,A -85,B 0,C 180,E1 -17483.926,E2 -17483.926} C_VEL
LIN {X 0,Y 277.261,Z 163.947,A -85,B 0,C 180,E1 -17487.482,E2 -17487.482} C_VEL
LIN {X 0,Y 277.242,Z 163.948,A -85,B 0,C 180,E1 -17490.474,E2 -17490.474} C_VEL
LIN {X 0,Y 277.24,Z 163.949,A -85,B 0,C 180,E1 -17493.897,E2 -17493.897} C_VEL
LIN {X 0,Y 277.249,Z 163.948,A -85,B 0,C 180,E1 -17497.473,E2 -17497.473} C_VEL
LIN {X 0,Y 277.179,Z 163.958,A -85,B 0,C 180,E1 -17501.242,E2 -17501.242} C_VEL
LIN {X 0,Y 277.194,Z 163.953,A -85,B 0,C 180,E1 -17505.228,E2 -17505.228} C_VEL
LIN {X 0,Y 277.215,Z 163.952,A -85,B 0,C 180,E1 -17509.514,E2 -17509.514} C_VEL
LIN {X 0,Y 277.254,Z 163.949,A -85,B 0,C 180,E1 -17512.53,E2 -17512.53} C_VEL
LIN {X 0,Y 277.243,Z 163.952,A -85,B 0,C 180,E1 -17516.105,E2 -17516.105} C_VEL
LIN {X 0,Y 277.279,Z 164.065,A -85,B 0,C 180,E1 -17519.606,E2 -17519.606} C_VEL
LIN {X 0,Y 277.83,Z 166.387,A -85,B 0,C 180,E1 -17520.504,E2 -17520.504} C_VEL
LIN {X 0,Y 287.015,Z 186.4,A -85,B 0,C 180,E1 -17522.111,E2 -17522.111} C_VEL
LIN {X 0,Y 292.657,Z 200.925,A -85,B 0,C 180,E1 -17523.094,E2 -17523.094} C_VEL
LIN {X 0,Y 290.659,Z 271.666,A -85,B 0,C 180,E1 -17524.825,E2 -17524.825} C_VEL
LIN {X 0,Y 289.868,Z 284.921,A -85,B 0,C 180,E1 -17525.374,E2 -17525.374} C_VEL
LIN {X 0,Y 288.735,Z 298.058,A -85,B 0,C 180,E1 -17526.226,E2 -17526.226} C_VEL
LIN {X 0,Y 287.231,Z 310.501,A -85,B 0,C 180,E1 -17527.334,E2 -17527.334} C_VEL
LIN {X 0,Y 285.512,Z 322.133,A -85,B 0,C 180,E1 -17528.712,E2 -17528.712} C_VEL
LIN {X 0,Y 283.891,Z 333.067,A -85,B 0,C 180,E1 -17530.377,E2 -17530.377} C_VEL
LIN {X 0,Y 282.44,Z 341.094,A -85,B 0,C 180,E1 -17531.879,E2 -17531.879} C_VEL
LIN {X 0,Y 280.84,Z 348.952,A -85,B 0,C 180,E1 -17533.649,E2 -17533.649} C_VEL
LIN {X 0,Y 279.245,Z 356.626,A -85,B 0,C 180,E1 -17535.796,E2 -17535.796} C_VEL
LIN {X 0,Y 277.757,Z 363.669,A -85,B 0,C 180,E1 -17538.322,E2 -17538.322} C_VEL
LIN {X 0,Y 276.79,Z 368.358,A -85,B 0,C 180,E1 -17540.501,E2 -17540.501} C_VEL
LIN {X 0,Y 276.079,Z 372.55,A -85,B 0,C 180,E1 -17543.124,E2 -17543.124} C_VEL
LIN {X 0,Y 275.691,Z 375.182,A -85,B 0,C 180,E1 -17545.615,E2 -17545.615} C_VEL
LIN {X 0,Y 275.363,Z 376.784,A -85,B 0,C 180,E1 -17548.538,E2 -17548.538} C_VEL
LIN {X 0,Y 275.342,Z 377.014,A -85,B 0,C 180,E1 -17550.001,E2 -17550.001} C_VEL
LIN {X 0,Y 275.363,Z 376.822,A -85,B 0,C 180,E1 -17551.463,E2 -17551.463} C_VEL
LIN {X 0,Y 275.683,Z 375.269,A -85,B 0,C 180,E1 -17554.387,E2 -17554.387} C_VEL
LIN {X 0,Y 276.106,Z 372.635,A -85,B 0,C 180,E1 -17556.922,E2 -17556.922} C_VEL
LIN {X 0,Y 276.75,Z 368.588,A -85,B 0,C 180,E1 -17559.502,E2 -17559.502} C_VEL
LIN {X 0,Y 277.708,Z 363.961,A -85,B 0,C 180,E1 -17561.681,E2 -17561.681} C_VEL
LIN {X 0,Y 279.199,Z 356.983,A -85,B 0,C 180,E1 -17564.208,E2 -17564.208} C_VEL
LIN {X 0,Y 280.736,Z 349.419,A -85,B 0,C 180,E1 -17566.358,E2 -17566.358} C_VEL
LIN {X 0,Y 282.706,Z 339.89,A -85,B 0,C 180,E1 -17568.48,E2 -17568.48} C_VEL
LIN {X 0,Y 284.378,Z 330.059,A -85,B 0,C 180,E1 -17570.243,E2 -17570.243} C_VEL
LIN {X 0,Y 285.922,Z 320.376,A -85,B 0,C 180,E1 -17571.636,E2 -17571.636} C_VEL
LIN {X 0,Y 287.394,Z 309.887,A -85,B 0,C 180,E1 -17572.844,E2 -17572.844} C_VEL
LIN {X 0,Y 288.756,Z 298.376,A -85,B 0,C 180,E1 -17573.869,E2 -17573.869} C_VEL
LIN {X 0,Y 289.92,Z 285.343,A -85,B 0,C 180,E1 -17574.719,E2 -17574.719} C_VEL
LIN {X 0,Y 290.763,Z 272.475,A -85,B 0,C 180,E1 -17575.263,E2 -17575.263} C_VEL
LIN {X 0,Y 292.664,Z 200.892,A -85,B 0,C 180,E1 -17577.03,E2 -17577.03} C_VEL
LIN {X 0,Y 285.963,Z 184,A -85,B 0,C 180,E1 -17578.196,E2 -17578.196} C_VEL
LIN {X 0,Y 279.145,Z 169.308,A -85,B 0,C 180,E1 -17579.381,E2 -17579.381} C_VEL
LIN {X 0,Y 277.806,Z 166.318,A -85,B 0,C 180,E1 -17579.656,E2 -17579.656} C_VEL
LIN {X 0,Y 277.25,Z 163.947,A -85,B 0,C 180,E1 -17580.653,E2 -17580.653} C_VEL
LIN {X 0,Y 277.248,Z 163.95,A -85,B 0,C 180,E1 -17583.896,E2 -17583.896} C_VEL
LIN {X 0,Y 277.25,Z 163.95,A -85,B 0,C 180,E1 -17587.472,E2 -17587.472} C_VEL
LIN {X 0,Y 277.178,Z 163.96,A -85,B 0,C 180,E1 -17591.242,E2 -17591.242} C_VEL
LIN {X 0,Y 277.175,Z 163.956,A -85,B 0,C 180,E1 -17595.232,E2 -17595.232} C_VEL
LIN {X 0,Y 277.185,Z 163.957,A -85,B 0,C 180,E1 -17598.759,E2 -17598.759} C_VEL
LIN {X 0,Y 277.255,Z 163.947,A -85,B 0,C 180,E1 -17602.528,E2 -17602.528} C_VEL
LIN {X 0,Y 277.246,Z 163.945,A -85,B 0,C 180,E1 -17606.104,E2 -17606.104} C_VEL
LIN {X 0,Y 277.262,Z 163.942,A -85,B 0,C 180,E1 -17609.538,E2 -17609.538} C_VEL
LIN {X 0,Y 277.292,Z 163.943,A -85,B 0,C 180,E1 -17612.857,E2 -17612.857} C_VEL
LIN {X 0,Y 277.285,Z 163.941,A -85,B 0,C 180,E1 -17616.075,E2 -17616.075} C_VEL
LIN {X 0,Y 277.254,Z 163.937,A -85,B 0,C 180,E1 -17617.931,E2 -17617.931} C_VEL
LIN {X 0,Y 276.576,Z 164.031,A -85,B 0,C 180,E1 -17619.143,E2 -17619.143} C_VEL
LIN {X 0,Y 273.755,Z 164.384,A -85,B 0,C 180,E1 -17621.12,E2 -17621.12} C_VEL
LIN {X 0,Y 271.385,Z 164.677,A -85,B 0,C 180,E1 -17622.726,E2 -17622.726} C_VEL
LIN {X 0,Y 270.388,Z 164.797,A -85,B 0,C 180,E1 -17623.97,E2 -17623.97} C_VEL
LIN {X 0,Y 270.315,Z 164.803,A -85,B 0,C 180,E1 -17624.391,E2 -17624.391} C_VEL
LIN {X 0,Y 270.367,Z 164.805,A -85,B 0,C 180,E1 -17627.997,E2 -17627.997} C_VEL
LIN {X 0,Y 270.528,Z 164.781,A -85,B 0,C 180,E1 -17631.032,E2 -17631.032} C_VEL
LIN {X 0,Y 270.506,Z 164.778,A -85,B 0,C 180,E1 -17634.035,E2 -17634.035} C_VEL
LIN {X 0,Y 270.768,Z 164.754,A -85,B 0,C 180,E1 -17638.513,E2 -17638.513} C_VEL
LIN {X 0,Y 270.766,Z 164.742,A -85,B 0,C 180,E1 -17641.487,E2 -17641.487} C_VEL
LIN {X 0,Y 270.551,Z 164.781,A -85,B 0,C 180,E1 -17647.463,E2 -17647.463} C_VEL
LIN {X 0,Y 270.38,Z 164.798,A -85,B 0,C 180,E1 -17650.483,E2 -17650.483} C_VEL
LIN {X 0,Y 270.335,Z 164.807,A -85,B 0,C 180,E1 -17655.068,E2 -17655.068} C_VEL
LIN {X 0,Y 270.214,Z 164.826,A -85,B 0,C 180,E1 -17659.762,E2 -17659.762} C_VEL
LIN {X 0,Y 270.181,Z 164.825,A -85,B 0,C 180,E1 -17664.436,E2 -17664.436} C_VEL
LIN {X 0,Y 270.195,Z 164.823,A -85,B 0,C 180,E1 -17667.917,E2 -17667.917} C_VEL
LIN {X 0,Y 270.173,Z 164.832,A -85,B 0,C 180,E1 -17671.35,E2 -17671.35} C_VEL
LIN {X 0,Y 270.198,Z 164.824,A -85,B 0,C 180,E1 -17674.906,E2 -17674.906} C_VEL
LIN {X 0,Y 270.198,Z 164.824,A -85,B 0,C 180,E1 -17678.71,E2 -17678.71} C_VEL
LIN {X 0,Y 270.148,Z 164.834,A -85,B 0,C 180,E1 -17683.245,E2 -17683.245} C_VEL
LIN {X 0,Y 270.151,Z 164.83,A -85,B 0,C 180,E1 -17687.437,E2 -17687.437} C_VEL
LIN {X 0,Y 270.208,Z 164.824,A -85,B 0,C 180,E1 -17691.374,E2 -17691.374} C_VEL
LIN {X 0,Y 270.251,Z 164.991,A -85,B 0,C 180,E1 -17693.206,E2 -17693.206} C_VEL
LIN {X 0,Y 272.573,Z 174.619,A -85,B 0,C 180,E1 -17696.83,E2 -17696.83} C_VEL
LIN {X 0,Y 274.518,Z 183.63,A -85,B 0,C 180,E1 -17700.024,E2 -17700.024} C_VEL
LIN {X 0,Y 280.129,Z 197.675,A -85,B 0,C 180,E1 -17701.08,E2 -17701.08} C_VEL
LIN {X 0,Y 284.245,Z 222.833,A -85,B 0,C 180,E1 -17702.237,E2 -17702.237} C_VEL
LIN {X 0,Y 285.518,Z 232.59,A -85,B 0,C 180,E1 -17702.641,E2 -17702.641} C_VEL
LIN {X 0,Y 283.742,Z 292.721,A -85,B 0,C 180,E1 -17704.165,E2 -17704.165} C_VEL
LIN {X 0,Y 282.684,Z 306.638,A -85,B 0,C 180,E1 -17704.801,E2 -17704.801} C_VEL
LIN {X 0,Y 281.188,Z 319.084,A -85,B 0,C 180,E1 -17705.644,E2 -17705.644} C_VEL
LIN {X 0,Y 279.615,Z 330.192,A -85,B 0,C 180,E1 -17706.679,E2 -17706.679} C_VEL
LIN {X 0,Y 277.697,Z 341.769,A -85,B 0,C 180,E1 -17708.081,E2 -17708.081} C_VEL
LIN {X 0,Y 275.715,Z 352.197,A -85,B 0,C 180,E1 -17709.677,E2 -17709.677} C_VEL
LIN {X 0,Y 274.05,Z 361.085,A -85,B 0,C 180,E1 -17711.38,E2 -17711.38} C_VEL
LIN {X 0,Y 272.299,Z 369.988,A -85,B 0,C 180,E1 -17713.506,E2 -17713.506} C_VEL
LIN {X 0,Y 270.771,Z 377.429,A -85,B 0,C 180,E1 -17715.724,E2 -17715.724} C_VEL
LIN {X 0,Y 269.569,Z 383.409,A -85,B 0,C 180,E1 -17717.961,E2 -17717.961} C_VEL
LIN {X 0,Y 268.873,Z 388.143,A -85,B 0,C 180,E1 -17720.217,E2 -17720.217} C_VEL
LIN {X 0,Y 268.37,Z 391.761,A -85,B 0,C 180,E1 -17722.475,E2 -17722.475} C_VEL
LIN {X 0,Y 268.171,Z 394.427,A -85,B 0,C 180,E1 -17724.794,E2 -17724.794} C_VEL
LIN {X 0,Y 268.193,Z 396.036,A -85,B 0,C 180,E1 -17726.995,E2 -17726.995} C_VEL
LIN {X 0,Y 268.219,Z 396.648,A -85,B 0,C 180,E1 -17728.498,E2 -17728.498} C_VEL
LIN {X 0,Y 268.251,Z 396.863,A -85,B 0,C 180,E1 -17729.999,E2 -17729.999} C_VEL
LIN {X 0,Y 268.219,Z 396.639,A -85,B 0,C 180,E1 -17731.501,E2 -17731.501} C_VEL
LIN {X 0,Y 268.193,Z 396.023,A -85,B 0,C 180,E1 -17733.003,E2 -17733.003} C_VEL
LIN {X 0,Y 268.176,Z 394.388,A -85,B 0,C 180,E1 -17735.218,E2 -17735.218} C_VEL
LIN {X 0,Y 268.534,Z 390.645,A -85,B 0,C 180,E1 -17738.275,E2 -17738.275} C_VEL
LIN {X 0,Y 269.073,Z 386.646,A -85,B 0,C 180,E1 -17740.534,E2 -17740.534} C_VEL
LIN {X 0,Y 270.089,Z 380.504,A -85,B 0,C 180,E1 -17743.16,E2 -17743.16} C_VEL
LIN {X 0,Y 271.532,Z 373.811,A -85,B 0,C 180,E1 -17745.384,E2 -17745.384} C_VEL
LIN {X 0,Y 273.227,Z 365.507,A -85,B 0,C 180,E1 -17747.591,E2 -17747.591} C_VEL
LIN {X 0,Y 274.766,Z 356.989,A -85,B 0,C 180,E1 -17749.42,E2 -17749.42} C_VEL
LIN {X 0,Y 276.787,Z 346.478,A -85,B 0,C 180,E1 -17751.211,E2 -17751.211} C_VEL
LIN {X 0,Y 278.863,Z 334.651,A -85,B 0,C 180,E1 -17752.797,E2 -17752.797} C_VEL
LIN {X 0,Y 280.638,Z 322.741,A -85,B 0,C 180,E1 -17754.012,E2 -17754.012} C_VEL
LIN {X 0,Y 282.184,Z 310.348,A -85,B 0,C 180,E1 -17754.95,E2 -17754.95} C_VEL
LIN {X 0,Y 283.37,Z 297.586,A -85,B 0,C 180,E1 -17755.624,E2 -17755.624} C_VEL
LIN {X 0,Y 284.018,Z 284.088,A -85,B 0,C 180,E1 -17756.053,E2 -17756.053} C_VEL
LIN {X 0,Y 285.389,Z 231.478,A -85,B 0,C 180,E1 -17757.368,E2 -17757.368} C_VEL
LIN {X 0,Y 281.144,Z 203.411,A -85,B 0,C 180,E1 -17758.606,E2 -17758.606} C_VEL
LIN {X 0,Y 279.615,Z 196.204,A -85,B 0,C 180,E1 -17758.981,E2 -17758.981} C_VEL
LIN {X 0,Y 274.463,Z 183.535,A -85,B 0,C 180,E1 -17759.97,E2 -17759.97} C_VEL
LIN {X 0,Y 272.273,Z 173.324,A -85,B 0,C 180,E1 -17763.6,E2 -17763.6} C_VEL
LIN {X 0,Y 270.228,Z 164.81,A -85,B 0,C 180,E1 -17766.854,E2 -17766.854} C_VEL
LIN {X 0,Y 270.141,Z 164.833,A -85,B 0,C 180,E1 -17771.021,E2 -17771.021} C_VEL
LIN {X 0,Y 270.124,Z 164.837,A -85,B 0,C 180,E1 -17774.624,E2 -17774.624} C_VEL
LIN {X 0,Y 270.146,Z 164.835,A -85,B 0,C 180,E1 -17777.437,E2 -17777.437} C_VEL
LIN {X 0,Y 270.202,Z 164.827,A -85,B 0,C 180,E1 -17781.373,E2 -17781.373} C_VEL
LIN {X 0,Y 270.192,Z 164.829,A -85,B 0,C 180,E1 -17785.093,E2 -17785.093} C_VEL
LIN {X 0,Y 270.178,Z 164.829,A -85,B 0,C 180,E1 -17789.136,E2 -17789.136} C_VEL
LIN {X 0,Y 270.193,Z 164.819,A -85,B 0,C 180,E1 -17792.172,E2 -17792.172} C_VEL
LIN {X 0,Y 270.175,Z 164.826,A -85,B 0,C 180,E1 -17795.563,E2 -17795.563} C_VEL
LIN {X 0,Y 270.212,Z 164.827,A -85,B 0,C 180,E1 -17800.238,E2 -17800.238} C_VEL
LIN {X 0,Y 270.33,Z 164.809,A -85,B 0,C 180,E1 -17804.931,E2 -17804.931} C_VEL
LIN {X 0,Y 270.376,Z 164.799,A -85,B 0,C 180,E1 -17809.516,E2 -17809.516} C_VEL
LIN {X 0,Y 270.544,Z 164.785,A -85,B 0,C 180,E1 -17812.537,E2 -17812.537} C_VEL
LIN {X 0,Y 270.759,Z 164.753,A -85,B 0,C 180,E1 -17818.513,E2 -17818.513} C_VEL
LIN {X 0,Y 270.761,Z 164.758,A -85,B 0,C 180,E1 -17821.487,E2 -17821.487} C_VEL
LIN {X 0,Y 270.554,Z 164.781,A -85,B 0,C 180,E1 -17827.463,E2 -17827.463} C_VEL
LIN {X 0,Y 270.378,Z 164.801,A -85,B 0,C 180,E1 -17830.484,E2 -17830.484} C_VEL
LIN {X 0,Y 270.33,Z 164.809,A -85,B 0,C 180,E1 -17835.069,E2 -17835.069} C_VEL
LIN {X 0,Y 270.215,Z 164.818,A -85,B 0,C 180,E1 -17839.762,E2 -17839.762} C_VEL
LIN {X 0,Y 270.211,Z 164.823,A -85,B 0,C 180,E1 -17844.453,E2 -17844.453} C_VEL
LIN {X 0,Y 270.19,Z 164.827,A -85,B 0,C 180,E1 -17847.918,E2 -17847.918} C_VEL
LIN {X 0,Y 270.168,Z 164.825,A -85,B 0,C 180,E1 -17851.351,E2 -17851.351} C_VEL
LIN {X 0,Y 270.192,Z 164.83,A -85,B 0,C 180,E1 -17854.907,E2 -17854.907} C_VEL
LIN {X 0,Y 270.193,Z 164.829,A -85,B 0,C 180,E1 -17858.711,E2 -17858.711} C_VEL
LIN {X 0,Y 270.144,Z 164.834,A -85,B 0,C 180,E1 -17863.246,E2 -17863.246} C_VEL
LIN {X 0,Y 270.159,Z 164.831,A -85,B 0,C 180,E1 -17867.441,E2 -17867.441} C_VEL
LIN {X 0,Y 270.204,Z 164.823,A -85,B 0,C 180,E1 -17871.375,E2 -17871.375} C_VEL
LIN {X 0,Y 270.196,Z 164.829,A -85,B 0,C 180,E1 -17875.095,E2 -17875.095} C_VEL
LIN {X 0,Y 270.216,Z 165.02,A -85,B 0,C 180,E1 -17878.968,E2 -17878.968} C_VEL
LIN {X 0,Y 270.626,Z 166.696,A -85,B 0,C 180,E1 -17879.641,E2 -17879.641} C_VEL
LIN {X 0,Y 279.077,Z 184.667,A -85,B 0,C 180,E1 -17881.185,E2 -17881.185} C_VEL
LIN {X 0,Y 284.879,Z 198.831,A -85,B 0,C 180,E1 -17882.229,E2 -17882.229} C_VEL
LIN {X 0,Y 286.307,Z 202.531,A -85,B 0,C 180,E1 -17882.484,E2 -17882.484} C_VEL
LIN {X 0,Y 284.265,Z 271.945,A -85,B 0,C 180,E1 -17884.217,E2 -17884.217} C_VEL
LIN {X 0,Y 283.458,Z 285.19,A -85,B 0,C 180,E1 -17884.778,E2 -17884.778} C_VEL
LIN {X 0,Y 282.368,Z 297.198,A -85,B 0,C 180,E1 -17885.558,E2 -17885.558} C_VEL
LIN {X 0,Y 280.965,Z 309.03,A -85,B 0,C 180,E1 -17886.605,E2 -17886.605} C_VEL
LIN {X 0,Y 279.376,Z 319.767,A -85,B 0,C 180,E1 -17887.832,E2 -17887.832} C_VEL
LIN {X 0,Y 277.785,Z 329.632,A -85,B 0,C 180,E1 -17889.257,E2 -17889.257} C_VEL
LIN {X 0,Y 276.114,Z 339.581,A -85,B 0,C 180,E1 -17891.064,E2 -17891.064} C_VEL
LIN {X 0,Y 274.322,Z 347.737,A -85,B 0,C 180,E1 -17892.866,E2 -17892.866} C_VEL
LIN {X 0,Y 272.592,Z 355.721,A -85,B 0,C 180,E1 -17895.06,E2 -17895.06} C_VEL
LIN {X 0,Y 271.212,Z 362.125,A -85,B 0,C 180,E1 -17897.277,E2 -17897.277} C_VEL
LIN {X 0,Y 270.092,Z 367.204,A -85,B 0,C 180,E1 -17899.506,E2 -17899.506} C_VEL
LIN {X 0,Y 269.299,Z 371.145,A -85,B 0,C 180,E1 -17901.748,E2 -17901.748} C_VEL
LIN {X 0,Y 268.826,Z 374.051,A -85,B 0,C 180,E1 -17903.998,E2 -17903.998} C_VEL
LIN {X 0,Y 268.617,Z 375.442,A -85,B 0,C 180,E1 -17905.499,E2 -17905.499} C_VEL
LIN {X 0,Y 268.289,Z 377.042,A -85,B 0,C 180,E1 -17908.5,E2 -17908.5} C_VEL
LIN {X 0,Y 268.264,Z 377.272,A -85,B 0,C 180,E1 -17910.001,E2 -17910.001} C_VEL
LIN {X 0,Y 268.289,Z 377.08,A -85,B 0,C 180,E1 -17911.502,E2 -17911.502} C_VEL
LIN {X 0,Y 268.424,Z 376.494,A -85,B 0,C 180,E1 -17913.002,E2 -17913.002} C_VEL
LIN {X 0,Y 268.61,Z 375.528,A -85,B 0,C 180,E1 -17914.503,E2 -17914.503} C_VEL
LIN {X 0,Y 269.031,Z 373.099,A -85,B 0,C 180,E1 -17916.93,E2 -17916.93} C_VEL
LIN {X 0,Y 269.745,Z 368.846,A -85,B 0,C 180,E1 -17919.751,E2 -17919.751} C_VEL
LIN {X 0,Y 270.766,Z 364.219,A -85,B 0,C 180,E1 -17921.985,E2 -17921.985} C_VEL
LIN {X 0,Y 272.323,Z 357.24,A -85,B 0,C 180,E1 -17924.574,E2 -17924.574} C_VEL
LIN {X 0,Y 273.942,Z 349.676,A -85,B 0,C 180,E1 -17926.776,E2 -17926.776} C_VEL
LIN {X 0,Y 275.634,Z 341.918,A -85,B 0,C 180,E1 -17928.586,E2 -17928.586} C_VEL
LIN {X 0,Y 277.284,Z 332.892,A -85,B 0,C 180,E1 -17930.315,E2 -17930.315} C_VEL
LIN {X 0,Y 279.13,Z 321.92,A -85,B 0,C 180,E1 -17931.995,E2 -17931.995} C_VEL
LIN {X 0,Y 280.882,Z 310.139,A -85,B 0,C 180,E1 -17933.404,E2 -17933.404} C_VEL
LIN {X 0,Y 282.291,Z 298.627,A -85,B 0,C 180,E1 -17934.45,E2 -17934.45} C_VEL
LIN {X 0,Y 283.504,Z 285.591,A -85,B 0,C 180,E1 -17935.317,E2 -17935.317} C_VEL
LIN {X 0,Y 284.369,Z 272.714,A -85,B 0,C 180,E1 -17935.872,E2 -17935.872} C_VEL
LIN {X 0,Y 286.333,Z 202.576,A -85,B 0,C 180,E1 -17937.638,E2 -17937.638} C_VEL
LIN {X 0,Y 279.245,Z 184.967,A -85,B 0,C 180,E1 -17938.917,E2 -17938.917} C_VEL
LIN {X 0,Y 273.243,Z 172.198,A -85,B 0,C 180,E1 -17940.001,E2 -17940.001} C_VEL
LIN {X 0,Y 270.612,Z 166.616,A -85,B 0,C 180,E1 -17940.525,E2 -17940.525} C_VEL
LIN {X 0,Y 270.215,Z 164.818,A -85,B 0,C 180,E1 -17941.268,E2 -17941.268} C_VEL
LIN {X 0,Y 270.199,Z 164.826,A -85,B 0,C 180,E1 -17944.906,E2 -17944.906} C_VEL
LIN {X 0,Y 270.169,Z 164.831,A -85,B 0,C 180,E1 -17948.702,E2 -17948.702} C_VEL
LIN {X 0,Y 270.149,Z 164.835,A -85,B 0,C 180,E1 -17953.245,E2 -17953.245} C_VEL
LIN {X 0,Y 270.152,Z 164.835,A -85,B 0,C 180,E1 -17957.438,E2 -17957.438} C_VEL
LIN {X 0,Y 270.208,Z 164.825,A -85,B 0,C 180,E1 -17961.374,E2 -17961.374} C_VEL
LIN {X 0,Y 270.198,Z 164.821,A -85,B 0,C 180,E1 -17965.094,E2 -17965.094} C_VEL
LIN {X 0,Y 270.185,Z 164.826,A -85,B 0,C 180,E1 -17969.136,E2 -17969.136} C_VEL
LIN {X 0,Y 270.223,Z 164.819,A -85,B 0,C 180,E1 -17972.163,E2 -17972.163} C_VEL
LIN {X 0,Y 270.229,Z 164.82,A -85,B 0,C 180,E1 -17975.542,E2 -17975.542} C_VEL
LIN {X 0,Y 270.249,Z 164.82,A -85,B 0,C 180,E1 -17980.24,E2 -17980.24} C_VEL
LIN {X 0,Y 270.315,Z 164.803,A -85,B 0,C 180,E1 -17984.391,E2 -17984.391} C_VEL
LIN {X 0,Y 269.69,Z 164.88,A -85,B 0,C 180,E1 -17985.634,E2 -17985.634} C_VEL
LIN {X 0,Y 266.927,Z 165.232,A -85,B 0,C 180,E1 -17987.661,E2 -17987.661} C_VEL
LIN {X 0,Y 264.566,Z 165.53,A -85,B 0,C 180,E1 -17989.31,E2 -17989.31} C_VEL
LIN {X 0,Y 263.551,Z 165.652,A -85,B 0,C 180,E1 -17990.585,E2 -17990.585} C_VEL
LIN {X 0,Y 263.468,Z 165.658,A -85,B 0,C 180,E1 -17991.017,E2 -17991.017} C_VEL
LIN {X 0,Y 263.479,Z 165.652,A -85,B 0,C 180,E1 -17993.875,E2 -17993.875} C_VEL
LIN {X 0,Y 263.732,Z 165.63,A -85,B 0,C 180,E1 -17998.473,E2 -17998.473} C_VEL
LIN {X 0,Y 263.73,Z 165.618,A -85,B 0,C 180,E1 -18001.527,E2 -18001.527} C_VEL
LIN {X 0,Y 263.513,Z 165.654,A -85,B 0,C 180,E1 -18007.663,E2 -18007.663} C_VEL
LIN {X 0,Y 263.325,Z 165.676,A -85,B 0,C 180,E1 -18010.768,E2 -18010.768} C_VEL
LIN {X 0,Y 263.287,Z 165.681,A -85,B 0,C 180,E1 -18015.482,E2 -18015.482} C_VEL
LIN {X 0,Y 263.205,Z 165.697,A -85,B 0,C 180,E1 -18020.311,E2 -18020.311} C_VEL
LIN {X 0,Y 263.125,Z 165.708,A -85,B 0,C 180,E1 -18025.3,E2 -18025.3} C_VEL
LIN {X 0,Y 263.129,Z 165.702,A -85,B 0,C 180,E1 -18028.736,E2 -18028.736} C_VEL
LIN {X 0,Y 263.128,Z 165.707,A -85,B 0,C 180,E1 -18032.289,E2 -18032.289} C_VEL
LIN {X 0,Y 263.175,Z 165.703,A -85,B 0,C 180,E1 -18036.761,E2 -18036.761} C_VEL
LIN {X 0,Y 263.092,Z 165.712,A -85,B 0,C 180,E1 -18039.875,E2 -18039.875} C_VEL
LIN {X 0,Y 263.077,Z 165.714,A -85,B 0,C 180,E1 -18043.994,E2 -18043.994} C_VEL
LIN {X 0,Y 263.081,Z 165.714,A -85,B 0,C 180,E1 -18048.417,E2 -18048.417} C_VEL
LIN {X 0,Y 263.194,Z 165.806,A -85,B 0,C 180,E1 -18052.461,E2 -18052.461} C_VEL
LIN {X 0,Y 265.168,Z 173.85,A -85,B 0,C 180,E1 -18055.619,E2 -18055.619} C_VEL
LIN {X 0,Y 267.296,Z 183.515,A -85,B 0,C 180,E1 -18059.132,E2 -18059.132} C_VEL
LIN {X 0,Y 274.142,Z 200.036,A -85,B 0,C 180,E1 -18060.463,E2 -18060.463} C_VEL
LIN {X 0,Y 278.03,Z 224.29,A -85,B 0,C 180,E1 -18061.61,E2 -18061.61} C_VEL
LIN {X 0,Y 279.205,Z 233.359,A -85,B 0,C 180,E1 -18061.997,E2 -18061.997} C_VEL
LIN {X 0,Y 277.389,Z 292.477,A -85,B 0,C 180,E1 -18063.528,E2 -18063.528} C_VEL
LIN {X 0,Y 276.275,Z 306.387,A -85,B 0,C 180,E1 -18064.174,E2 -18064.174} C_VEL
LIN {X 0,Y 274.745,Z 318.831,A -85,B 0,C 180,E1 -18065.034,E2 -18065.034} C_VEL
LIN {X 0,Y 273.112,Z 329.937,A -85,B 0,C 180,E1 -18066.09,E2 -18066.09} C_VEL
LIN {X 0,Y 271.102,Z 341.513,A -85,B 0,C 180,E1 -18067.519,E2 -18067.519} C_VEL
LIN {X 0,Y 269.051,Z 351.94,A -85,B 0,C 180,E1 -18069.151,E2 -18069.151} C_VEL
LIN {X 0,Y 267.36,Z 360.474,A -85,B 0,C 180,E1 -18070.817,E2 -18070.817} C_VEL
LIN {X 0,Y 265.783,Z 368.52,A -85,B 0,C 180,E1 -18072.739,E2 -18072.739} C_VEL
LIN {X 0,Y 264.142,Z 376.049,A -85,B 0,C 180,E1 -18074.964,E2 -18074.964} C_VEL
LIN {X 0,Y 262.584,Z 383.149,A -85,B 0,C 180,E1 -18077.636,E2 -18077.636} C_VEL
LIN {X 0,Y 261.83,Z 387.883,A -85,B 0,C 180,E1 -18079.951,E2 -18079.951} C_VEL
LIN {X 0,Y 261.314,Z 391.502,A -85,B 0,C 180,E1 -18082.271,E2 -18082.271} C_VEL
LIN {X 0,Y 261.086,Z 394.367,A -85,B 0,C 180,E1 -18084.862,E2 -18084.862} C_VEL
LIN {X 0,Y 261.104,Z 395.778,A -85,B 0,C 180,E1 -18086.913,E2 -18086.913} C_VEL
LIN {X 0,Y 261.145,Z 396.39,A -85,B 0,C 180,E1 -18088.457,E2 -18088.457} C_VEL
LIN {X 0,Y 261.175,Z 396.605,A -85,B 0,C 180,E1 -18089.999,E2 -18089.999} C_VEL
LIN {X 0,Y 261.145,Z 396.381,A -85,B 0,C 180,E1 -18091.541,E2 -18091.541} C_VEL
LIN {X 0,Y 261.105,Z 395.763,A -85,B 0,C 180,E1 -18093.085,E2 -18093.085} C_VEL
LIN {X 0,Y 261.085,Z 394.341,A -85,B 0,C 180,E1 -18095.136,E2 -18095.136} C_VEL
LIN {X 0,Y 261.333,Z 391.462,A -85,B 0,C 180,E1 -18097.727,E2 -18097.727} C_VEL
LIN {X 0,Y 261.829,Z 387.824,A -85,B 0,C 180,E1 -18100.047,E2 -18100.047} C_VEL
LIN {X 0,Y 262.583,Z 383.073,A -85,B 0,C 180,E1 -18102.363,E2 -18102.363} C_VEL
LIN {X 0,Y 264.139,Z 375.956,A -85,B 0,C 180,E1 -18105.035,E2 -18105.035} C_VEL
LIN {X 0,Y 265.788,Z 368.373,A -85,B 0,C 180,E1 -18107.266,E2 -18107.266} C_VEL
LIN {X 0,Y 267.344,Z 360.322,A -85,B 0,C 180,E1 -18109.183,E2 -18109.183} C_VEL
LIN {X 0,Y 269.262,Z 350.683,A -85,B 0,C 180,E1 -18111.031,E2 -18111.031} C_VEL
LIN {X 0,Y 271.336,Z 339.997,A -85,B 0,C 180,E1 -18112.66,E2 -18112.66} C_VEL
LIN {X 0,Y 273.074,Z 329.664,A -85,B 0,C 180,E1 -18113.912,E2 -18113.912} C_VEL
LIN {X 0,Y 274.883,Z 317.318,A -85,B 0,C 180,E1 -18115.052,E2 -18115.052} C_VEL
LIN {X 0,Y 276.385,Z 304.319,A -85,B 0,C 180,E1 -18115.914,E2 -18115.914} C_VEL
LIN {X 0,Y 277.33,Z 291.651,A -85,B 0,C 180,E1 -18116.477,E2 -18116.477} C_VEL
LIN {X 0,Y 279.069,Z 232.336,A -85,B 0,C 180,E1 -18118.009,E2 -18118.009} C_VEL
LIN {X 0,Y 274.865,Z 204.506,A -85,B 0,C 180,E1 -18119.282,E2 -18119.282} C_VEL
LIN {X 0,Y 273.57,Z 198.631,A -85,B 0,C 180,E1 -18119.605,E2 -18119.605} C_VEL
LIN {X 0,Y 268.086,Z 185.618,A -85,B 0,C 180,E1 -18120.661,E2 -18120.661} C_VEL
LIN {X 0,Y 267.201,Z 183.127,A -85,B 0,C 180,E1 -18120.906,E2 -18120.906} C_VEL
LIN {X 0,Y 264.927,Z 172.963,A -85,B 0,C 180,E1 -18124.677,E2 -18124.677} C_VEL
LIN {X 0,Y 263.171,Z 165.69,A -85,B 0,C 180,E1 -18127.578,E2 -18127.578} C_VEL
LIN {X 0,Y 263.076,Z 165.711,A -85,B 0,C 180,E1 -18131.901,E2 -18131.901} C_VEL
LIN {X 0,Y 263.074,Z 165.714,A -85,B 0,C 180,E1 -18136.16,E2 -18136.16} C_VEL
LIN {X 0,Y 263.107,Z 165.711,A -85,B 0,C 180,E1 -18140.77,E2 -18140.77} C_VEL
LIN {X 0,Y 263.151,Z 165.703,A -85,B 0,C 180,E1 -18144.016,E2 -18144.016} C_VEL
LIN {X 0,Y 263.122,Z 165.704,A -85,B 0,C 180,E1 -18147.71,E2 -18147.71} C_VEL
LIN {X 0,Y 263.14,Z 165.696,A -85,B 0,C 180,E1 -18151.805,E2 -18151.805} C_VEL
LIN {X 0,Y 263.108,Z 165.705,A -85,B 0,C 180,E1 -18156.38,E2 -18156.38} C_VEL
LIN {X 0,Y 263.2,Z 165.698,A -85,B 0,C 180,E1 -18159.688,E2 -18159.688} C_VEL
LIN {X 0,Y 263.28,Z 165.683,A -85,B 0,C 180,E1 -18164.518,E2 -18164.518} C_VEL
LIN {X 0,Y 263.321,Z 165.677,A -85,B 0,C 180,E1 -18169.232,E2 -18169.232} C_VEL
LIN {X 0,Y 263.506,Z 165.66,A -85,B 0,C 180,E1 -18172.336,E2 -18172.336} C_VEL
LIN {X 0,Y 263.722,Z 165.628,A -85,B 0,C 180,E1 -18178.473,E2 -18178.473} C_VEL
LIN {X 0,Y 263.725,Z 165.634,A -85,B 0,C 180,E1 -18181.527,E2 -18181.527} C_VEL
LIN {X 0,Y 263.518,Z 165.659,A -85,B 0,C 180,E1 -18187.663,E2 -18187.663} C_VEL
LIN {X 0,Y 263.322,Z 165.68,A -85,B 0,C 180,E1 -18190.768,E2 -18190.768} C_VEL
LIN {X 0,Y 263.28,Z 165.69,A -85,B 0,C 180,E1 -18195.482,E2 -18195.482} C_VEL
LIN {X 0,Y 263.203,Z 165.692,A -85,B 0,C 180,E1 -18200.312,E2 -18200.312} C_VEL
LIN {X 0,Y 263.149,Z 165.703,A -85,B 0,C 180,E1 -18204.767,E2 -18204.767} C_VEL
LIN {X 0,Y 263.127,Z 165.708,A -85,B 0,C 180,E1 -18208.736,E2 -18208.736} C_VEL
LIN {X 0,Y 263.122,Z 165.702,A -85,B 0,C 180,E1 -18212.29,E2 -18212.29} C_VEL
LIN {X 0,Y 263.17,Z 165.705,A -85,B 0,C 180,E1 -18216.762,E2 -18216.762} C_VEL
LIN {X 0,Y 263.086,Z 165.711,A -85,B 0,C 180,E1 -18219.876,E2 -18219.876} C_VEL
LIN {X 0,Y 263.094,Z 165.711,A -85,B 0,C 180,E1 -18223.991,E2 -18223.991} C_VEL
LIN {X 0,Y 263.116,Z 165.707,A -85,B 0,C 180,E1 -18228.409,E2 -18228.409} C_VEL
LIN {X 0,Y 263.154,Z 165.702,A -85,B 0,C 180,E1 -18232.104,E2 -18232.104} C_VEL
LIN {X 0,Y 263.149,Z 165.707,A -85,B 0,C 180,E1 -18235.887,E2 -18235.887} C_VEL
LIN {X 0,Y 263.12,Z 165.79,A -85,B 0,C 180,E1 -18238.216,E2 -18238.216} C_VEL
LIN {X 0,Y 263.42,Z 167.017,A -85,B 0,C 180,E1 -18238.72,E2 -18238.72} C_VEL
LIN {X 0,Y 272.197,Z 185.221,A -85,B 0,C 180,E1 -18240.392,E2 -18240.392} C_VEL
LIN {X 0,Y 278.566,Z 200.439,A -85,B 0,C 180,E1 -18241.581,E2 -18241.581} C_VEL
LIN {X 0,Y 280.05,Z 204.945,A -85,B 0,C 180,E1 -18241.876,E2 -18241.876} C_VEL
LIN {X 0,Y 277.852,Z 273.634,A -85,B 0,C 180,E1 -18243.627,E2 -18243.627} C_VEL
LIN {X 0,Y 276.948,Z 286.979,A -85,B 0,C 180,E1 -18244.243,E2 -18244.243} C_VEL
LIN {X 0,Y 275.713,Z 299.717,A -85,B 0,C 180,E1 -18245.129,E2 -18245.129} C_VEL
LIN {X 0,Y 274.225,Z 311.029,A -85,B 0,C 180,E1 -18246.195,E2 -18246.195} C_VEL
LIN {X 0,Y 272.371,Z 322.659,A -85,B 0,C 180,E1 -18247.631,E2 -18247.631} C_VEL
LIN {X 0,Y 270.755,Z 332.297,A -85,B 0,C 180,E1 -18249.141,E2 -18249.141} C_VEL
LIN {X 0,Y 269.029,Z 341.617,A -85,B 0,C 180,E1 -18250.942,E2 -18250.942} C_VEL
LIN {X 0,Y 267.222,Z 349.476,A -85,B 0,C 180,E1 -18252.791,E2 -18252.791} C_VEL
LIN {X 0,Y 265.507,Z 357.148,A -85,B 0,C 180,E1 -18255.045,E2 -18255.045} C_VEL
LIN {X 0,Y 263.88,Z 364.19,A -85,B 0,C 180,E1 -18257.699,E2 -18257.699} C_VEL
LIN {X 0,Y 262.805,Z 368.878,A -85,B 0,C 180,E1 -18259.991,E2 -18259.991} C_VEL
LIN {X 0,Y 262.08,Z 372.462,A -85,B 0,C 180,E1 -18262.295,E2 -18262.295} C_VEL
LIN {X 0,Y 261.76,Z 374.311,A -85,B 0,C 180,E1 -18263.836,E2 -18263.836} C_VEL
LIN {X 0,Y 261.547,Z 375.701,A -85,B 0,C 180,E1 -18265.377,E2 -18265.377} C_VEL
LIN {X 0,Y 261.363,Z 376.691,A -85,B 0,C 180,E1 -18266.918,E2 -18266.918} C_VEL
LIN {X 0,Y 261.188,Z 377.53,A -85,B 0,C 180,E1 -18270.001,E2 -18270.001} C_VEL
LIN {X 0,Y 261.217,Z 377.338,A -85,B 0,C 180,E1 -18271.543,E2 -18271.543} C_VEL
LIN {X 0,Y 261.361,Z 376.752,A -85,B 0,C 180,E1 -18273.084,E2 -18273.084} C_VEL
LIN {X 0,Y 261.54,Z 375.786,A -85,B 0,C 180,E1 -18274.625,E2 -18274.625} C_VEL
LIN {X 0,Y 261.953,Z 373.566,A -85,B 0,C 180,E1 -18276.934,E2 -18276.934} C_VEL
LIN {X 0,Y 262.504,Z 370.381,A -85,B 0,C 180,E1 -18279.245,E2 -18279.245} C_VEL
LIN {X 0,Y 263.422,Z 366.136,A -85,B 0,C 180,E1 -18281.543,E2 -18281.543} C_VEL
LIN {X 0,Y 264.926,Z 359.703,A -85,B 0,C 180,E1 -18284.205,E2 -18284.205} C_VEL
LIN {X 0,Y 266.516,Z 352.632,A -85,B 0,C 180,E1 -18286.468,E2 -18286.468} C_VEL
LIN {X 0,Y 268.547,Z 343.816,A -85,B 0,C 180,E1 -18288.699,E2 -18288.699} C_VEL
LIN {X 0,Y 270.245,Z 335.677,A -85,B 0,C 180,E1 -18290.368,E2 -18290.368} C_VEL
LIN {X 0,Y 271.885,Z 325.968,A -85,B 0,C 180,E1 -18292.013,E2 -18292.013} C_VEL
LIN {X 0,Y 273.708,Z 315.169,A -85,B 0,C 180,E1 -18293.453,E2 -18293.453} C_VEL
LIN {X 0,Y 275.411,Z 303.045,A -85,B 0,C 180,E1 -18294.7,E2 -18294.7} C_VEL
LIN {X 0,Y 276.78,Z 290.332,A -85,B 0,C 180,E1 -18295.674,E2 -18295.674} C_VEL
LIN {X 0,Y 277.722,Z 277.618,A -85,B 0,C 180,E1 -18296.337,E2 -18296.337} C_VEL
LIN {X 0,Y 278.514,Z 259.582,A -85,B 0,C 180,E1 -18296.862,E2 -18296.862} C_VEL
LIN {X 0,Y 280.065,Z 204.296,A -85,B 0,C 180,E1 -18298.269,E2 -18298.269} C_VEL
LIN {X 0,Y 272.757,Z 186.357,A -85,B 0,C 180,E1 -18299.638,E2 -18299.638} C_VEL
LIN {X 0,Y 265.105,Z 170.406,A -85,B 0,C 180,E1 -18301.087,E2 -18301.087} C_VEL
LIN {X 0,Y 263.433,Z 166.936,A -85,B 0,C 180,E1 -18301.44,E2 -18301.44} C_VEL
LIN {X 0,Y 263.142,Z 165.699,A -85,B 0,C 180,E1 -18302.002,E2 -18302.002} C_VEL
LIN {X 0,Y 263.158,Z 165.704,A -85,B 0,C 180,E1 -18305.983,E2 -18305.983} C_VEL
LIN {X 0,Y 263.074,Z 165.715,A -85,B 0,C 180,E1 -18309.879,E2 -18309.879} C_VEL
LIN {X 0,Y 263.077,Z 165.714,A -85,B 0,C 180,E1 -18313.994,E2 -18313.994} C_VEL
LIN {X 0,Y 263.081,Z 165.712,A -85,B 0,C 180,E1 -18318.417,E2 -18318.417} C_VEL
LIN {X 0,Y 263.158,Z 165.703,A -85,B 0,C 180,E1 -18322.102,E2 -18322.102} C_VEL
LIN {X 0,Y 263.152,Z 165.7,A -85,B 0,C 180,E1 -18325.885,E2 -18325.885} C_VEL
LIN {X 0,Y 263.126,Z 165.703,A -85,B 0,C 180,E1 -18329.503,E2 -18329.503} C_VEL
LIN {X 0,Y 263.143,Z 165.707,A -85,B 0,C 180,E1 -18332.997,E2 -18332.997} C_VEL
LIN {X 0,Y 263.148,Z 165.699,A -85,B 0,C 180,E1 -18336.383,E2 -18336.383} C_VEL
LIN {X 0,Y 263.235,Z 165.692,A -85,B 0,C 180,E1 -18339.691,E2 -18339.691} C_VEL
LIN {X 0,Y 263.288,Z 165.676,A -85,B 0,C 180,E1 -18344.518,E2 -18344.518} C_VEL
LIN {X 0,Y 263.347,Z 165.68,A -85,B 0,C 180,E1 -18349.233,E2 -18349.233} C_VEL
LIN {X 0,Y 263.468,Z 165.658,A -85,B 0,C 180,E1 -18351.017,E2 -18351.017} C_VEL
LIN {X 0,Y 262.778,Z 165.74,A -85,B 0,C 180,E1 -18352.292,E2 -18352.292} C_VEL
LIN {X 0,Y 259.874,Z 166.104,A -85,B 0,C 180,E1 -18354.369,E2 -18354.369} C_VEL
LIN {X 0,Y 257.495,Z 166.409,A -85,B 0,C 180,E1 -18356.06,E2 -18356.06} C_VEL
LIN {X 0,Y 256.588,Z 166.522,A -85,B 0,C 180,E1 -18357.371,E2 -18357.371} C_VEL
LIN {X 0,Y 256.574,Z 166.52,A -85,B 0,C 180,E1 -18357.814,E2 -18357.814} C_VEL
LIN {X 0,Y 256.692,Z 166.494,A -85,B 0,C 180,E1 -18361.569,E2 -18361.569} C_VEL
LIN {X 0,Y 256.449,Z 166.538,A -85,B 0,C 180,E1 -18366.293,E2 -18366.293} C_VEL
LIN {X 0,Y 256.398,Z 166.532,A -85,B 0,C 180,E1 -18369.466,E2 -18369.466} C_VEL
LIN {X 0,Y 256.194,Z 166.568,A -85,B 0,C 180,E1 -18374.294,E2 -18374.294} C_VEL
LIN {X 0,Y 256.139,Z 166.568,A -85,B 0,C 180,E1 -18377.567,E2 -18377.567} C_VEL
LIN {X 0,Y 256.118,Z 166.582,A -85,B 0,C 180,E1 -18381.096,E2 -18381.096} C_VEL
LIN {X 0,Y 256.084,Z 166.583,A -85,B 0,C 180,E1 -18385.088,E2 -18385.088} C_VEL
LIN {X 0,Y 256.086,Z 166.579,A -85,B 0,C 180,E1 -18388.573,E2 -18388.573} C_VEL
LIN {X 0,Y 256.074,Z 166.587,A -85,B 0,C 180,E1 -18391.701,E2 -18391.701} C_VEL
LIN {X 0,Y 256.08,Z 166.585,A -85,B 0,C 180,E1 -18395.193,E2 -18395.193} C_VEL
LIN {X 0,Y 256.066,Z 166.587,A -85,B 0,C 180,E1 -18399.143,E2 -18399.143} C_VEL
LIN {X 0,Y 256.023,Z 166.594,A -85,B 0,C 180,E1 -18403.335,E2 -18403.335} C_VEL
LIN {X 0,Y 256.034,Z 166.589,A -85,B 0,C 180,E1 -18407.828,E2 -18407.828} C_VEL
LIN {X 0,Y 256.135,Z 166.704,A -85,B 0,C 180,E1 -18411.698,E2 -18411.698} C_VEL
LIN {X 0,Y 258.261,Z 175.157,A -85,B 0,C 180,E1 -18415.147,E2 -18415.147} C_VEL
LIN {X 0,Y 260.046,Z 183.131,A -85,B 0,C 180,E1 -18418.169,E2 -18418.169} C_VEL
LIN {X 0,Y 267.828,Z 201.63,A -85,B 0,C 180,E1 -18419.75,E2 -18419.75} C_VEL
LIN {X 0,Y 269.419,Z 209.785,A -85,B 0,C 180,E1 -18420.19,E2 -18420.19} C_VEL
LIN {X 0,Y 272.897,Z 233.742,A -85,B 0,C 180,E1 -18421.309,E2 -18421.309} C_VEL
LIN {X 0,Y 271.064,Z 292.231,A -85,B 0,C 180,E1 -18422.86,E2 -18422.86} C_VEL
LIN {X 0,Y 269.986,Z 305.375,A -85,B 0,C 180,E1 -18423.474,E2 -18423.474} C_VEL
LIN {X 0,Y 268.474,Z 317.467,A -85,B 0,C 180,E1 -18424.305,E2 -18424.305} C_VEL
LIN {X 0,Y 266.641,Z 329.683,A -85,B 0,C 180,E1 -18425.472,E2 -18425.472} C_VEL
LIN {X 0,Y 264.537,Z 341.257,A -85,B 0,C 180,E1 -18426.929,E2 -18426.929} C_VEL
LIN {X 0,Y 262.426,Z 351.684,A -85,B 0,C 180,E1 -18428.599,E2 -18428.599} C_VEL
LIN {X 0,Y 260.632,Z 360.216,A -85,B 0,C 180,E1 -18430.301,E2 -18430.301} C_VEL
LIN {X 0,Y 258.954,Z 368.434,A -85,B 0,C 180,E1 -18432.319,E2 -18432.319} C_VEL
LIN {X 0,Y 257.268,Z 375.79,A -85,B 0,C 180,E1 -18434.552,E2 -18434.552} C_VEL
LIN {X 0,Y 255.606,Z 382.89,A -85,B 0,C 180,E1 -18437.292,E2 -18437.292} C_VEL
LIN {X 0,Y 254.797,Z 387.624,A -85,B 0,C 180,E1 -18439.671,E2 -18439.671} C_VEL
LIN {X 0,Y 254.255,Z 391.243,A -85,B 0,C 180,E1 -18442.055,E2 -18442.055} C_VEL
LIN {X 0,Y 253.984,Z 394.327,A -85,B 0,C 180,E1 -18444.978,E2 -18444.978} C_VEL
LIN {X 0,Y 253.999,Z 395.518,A -85,B 0,C 180,E1 -18446.827,E2 -18446.827} C_VEL
LIN {X 0,Y 254.072,Z 396.132,A -85,B 0,C 180,E1 -18448.414,E2 -18448.414} C_VEL
LIN {X 0,Y 254.1,Z 396.346,A -85,B 0,C 180,E1 -18449.999,E2 -18449.999} C_VEL
LIN {X 0,Y 254.072,Z 396.122,A -85,B 0,C 180,E1 -18451.584,E2 -18451.584} C_VEL
LIN {X 0,Y 253.999,Z 395.503,A -85,B 0,C 180,E1 -18453.171,E2 -18453.171} C_VEL
LIN {X 0,Y 253.983,Z 394.305,A -85,B 0,C 180,E1 -18455.02,E2 -18455.02} C_VEL
LIN {X 0,Y 254.295,Z 391.202,A -85,B 0,C 180,E1 -18457.942,E2 -18457.942} C_VEL
LIN {X 0,Y 254.797,Z 387.562,A -85,B 0,C 180,E1 -18460.327,E2 -18460.327} C_VEL
LIN {X 0,Y 255.604,Z 382.811,A -85,B 0,C 180,E1 -18462.706,E2 -18462.706} C_VEL
LIN {X 0,Y 257.262,Z 375.694,A -85,B 0,C 180,E1 -18465.446,E2 -18465.446} C_VEL
LIN {X 0,Y 258.952,Z 368.295,A -85,B 0,C 180,E1 -18467.685,E2 -18467.685} C_VEL
LIN {X 0,Y 260.621,Z 360.059,A -85,B 0,C 180,E1 -18469.698,E2 -18469.698} C_VEL
LIN {X 0,Y 262.614,Z 350.42,A -85,B 0,C 180,E1 -18471.589,E2 -18471.589} C_VEL
LIN {X 0,Y 264.784,Z 339.733,A -85,B 0,C 180,E1 -18473.253,E2 -18473.253} C_VEL
LIN {X 0,Y 266.599,Z 329.4,A -85,B 0,C 180,E1 -18474.53,E2 -18474.53} C_VEL
LIN {X 0,Y 268.468,Z 317.052,A -85,B 0,C 180,E1 -18475.693,E2 -18475.693} C_VEL
LIN {X 0,Y 270.028,Z 304.051,A -85,B 0,C 180,E1 -18476.572,E2 -18476.572} C_VEL
LIN {X 0,Y 271,Z 291.377,A -85,B 0,C 180,E1 -18477.145,E2 -18477.145} C_VEL
LIN {X 0,Y 272.801,Z 233.103,A -85,B 0,C 180,E1 -18478.681,E2 -18478.681} C_VEL
LIN {X 0,Y 268.54,Z 204.957,A -85,B 0,C 180,E1 -18480.019,E2 -18480.019} C_VEL
LIN {X 0,Y 267.559,Z 200.955,A -85,B 0,C 180,E1 -18480.261,E2 -18480.261} C_VEL
LIN {X 0,Y 261.241,Z 186.136,A -85,B 0,C 180,E1 -18481.529,E2 -18481.529} C_VEL
LIN {X 0,Y 259.937,Z 182.834,A -85,B 0,C 180,E1 -18481.864,E2 -18481.864} C_VEL
LIN {X 0,Y 257.992,Z 174.194,A -85,B 0,C 180,E1 -18485.191,E2 -18485.191} C_VEL
LIN {X 0,Y 256.097,Z 166.577,A -85,B 0,C 180,E1 -18488.342,E2 -18488.342} C_VEL
LIN {X 0,Y 256.03,Z 166.59,A -85,B 0,C 180,E1 -18492.171,E2 -18492.171} C_VEL
LIN {X 0,Y 256.017,Z 166.592,A -85,B 0,C 180,E1 -18496.663,E2 -18496.663} C_VEL
LIN {X 0,Y 256.061,Z 166.589,A -85,B 0,C 180,E1 -18500.856,E2 -18500.856} C_VEL
LIN {X 0,Y 256.12,Z 166.578,A -85,B 0,C 180,E1 -18502.866,E2 -18502.866} C_VEL
LIN {X 0,Y 256.06,Z 166.583,A -85,B 0,C 180,E1 -18506.706,E2 -18506.706} C_VEL
LIN {X 0,Y 256.048,Z 166.588,A -85,B 0,C 180,E1 -18510.392,E2 -18510.392} C_VEL
LIN {X 0,Y 256.067,Z 166.585,A -85,B 0,C 180,E1 -18513.951,E2 -18513.951} C_VEL
LIN {X 0,Y 256.049,Z 166.58,A -85,B 0,C 180,E1 -18517.402,E2 -18517.402} C_VEL
LIN {X 0,Y 256.099,Z 166.584,A -85,B 0,C 180,E1 -18520.773,E2 -18520.773} C_VEL
LIN {X 0,Y 256.205,Z 166.56,A -85,B 0,C 180,E1 -18524.079,E2 -18524.079} C_VEL
LIN {X 0,Y 256.265,Z 166.556,A -85,B 0,C 180,E1 -18528.932,E2 -18528.932} C_VEL
LIN {X 0,Y 256.447,Z 166.537,A -85,B 0,C 180,E1 -18532.124,E2 -18532.124} C_VEL
LIN {X 0,Y 256.434,Z 166.53,A -85,B 0,C 180,E1 -18536.858,E2 -18536.858} C_VEL
LIN {X 0,Y 256.685,Z 166.503,A -85,B 0,C 180,E1 -18538.431,E2 -18538.431} C_VEL
LIN {X 0,Y 256.687,Z 166.511,A -85,B 0,C 180,E1 -18541.569,E2 -18541.569} C_VEL
LIN {X 0,Y 256.438,Z 166.535,A -85,B 0,C 180,E1 -18546.576,E2 -18546.576} C_VEL
LIN {X 0,Y 256.395,Z 166.549,A -85,B 0,C 180,E1 -18549.466,E2 -18549.466} C_VEL
LIN {X 0,Y 256.194,Z 166.569,A -85,B 0,C 180,E1 -18554.294,E2 -18554.294} C_VEL
LIN {X 0,Y 256.142,Z 166.575,A -85,B 0,C 180,E1 -18557.567,E2 -18557.567} C_VEL
LIN {X 0,Y 256.117,Z 166.576,A -85,B 0,C 180,E1 -18561.1,E2 -18561.1} C_VEL
LIN {X 0,Y 256.098,Z 166.578,A -85,B 0,C 180,E1 -18565.099,E2 -18565.099} C_VEL
LIN {X 0,Y 256.083,Z 166.585,A -85,B 0,C 180,E1 -18568.576,E2 -18568.576} C_VEL
LIN {X 0,Y 256.068,Z 166.58,A -85,B 0,C 180,E1 -18571.702,E2 -18571.702} C_VEL
LIN {X 0,Y 256.074,Z 166.587,A -85,B 0,C 180,E1 -18575.194,E2 -18575.194} C_VEL
LIN {X 0,Y 256.104,Z 166.582,A -85,B 0,C 180,E1 -18577.27,E2 -18577.27} C_VEL
LIN {X 0,Y 256.014,Z 166.594,A -85,B 0,C 180,E1 -18581.212,E2 -18581.212} C_VEL
LIN {X 0,Y 256.035,Z 166.588,A -85,B 0,C 180,E1 -18585.536,E2 -18585.536} C_VEL
LIN {X 0,Y 256.047,Z 166.587,A -85,B 0,C 180,E1 -18588.797,E2 -18588.797} C_VEL
LIN {X 0,Y 256.124,Z 166.583,A -85,B 0,C 180,E1 -18592.868,E2 -18592.868} C_VEL
LIN {X 0,Y 256.086,Z 166.586,A -85,B 0,C 180,E1 -18597.356,E2 -18597.356} C_VEL
LIN {X 0,Y 256.272,Z 167.488,A -85,B 0,C 180,E1 -18597.748,E2 -18597.748} C_VEL
LIN {X 0,Y 257.799,Z 170.519,A -85,B 0,C 180,E1 -18598.062,E2 -18598.062} C_VEL
LIN {X 0,Y 265.045,Z 185.151,A -85,B 0,C 180,E1 -18599.497,E2 -18599.497} C_VEL
LIN {X 0,Y 271.729,Z 200.785,A -85,B 0,C 180,E1 -18600.799,E2 -18600.799} C_VEL
LIN {X 0,Y 273.655,Z 205.911,A -85,B 0,C 180,E1 -18601.178,E2 -18601.178} C_VEL
LIN {X 0,Y 271.645,Z 271,A -85,B 0,C 180,E1 -18602.872,E2 -18602.872} C_VEL
LIN {X 0,Y 270.834,Z 284.099,A -85,B 0,C 180,E1 -18603.41,E2 -18603.41} C_VEL
LIN {X 0,Y 269.66,Z 296.604,A -85,B 0,C 180,E1 -18604.221,E2 -18604.221} C_VEL
LIN {X 0,Y 268.308,Z 307.796,A -85,B 0,C 180,E1 -18605.224,E2 -18605.224} C_VEL
LIN {X 0,Y 266.562,Z 318.872,A -85,B 0,C 180,E1 -18606.5,E2 -18606.5} C_VEL
LIN {X 0,Y 264.744,Z 329.005,A -85,B 0,C 180,E1 -18607.979,E2 -18607.979} C_VEL
LIN {X 0,Y 263.139,Z 338.301,A -85,B 0,C 180,E1 -18609.685,E2 -18609.685} C_VEL
LIN {X 0,Y 261.182,Z 346.781,A -85,B 0,C 180,E1 -18611.569,E2 -18611.569} C_VEL
LIN {X 0,Y 259.184,Z 355.021,A -85,B 0,C 180,E1 -18613.864,E2 -18613.864} C_VEL
LIN {X 0,Y 257.829,Z 360.653,A -85,B 0,C 180,E1 -18615.8,E2 -18615.8} C_VEL
LIN {X 0,Y 256.526,Z 366.141,A -85,B 0,C 180,E1 -18618.144,E2 -18618.144} C_VEL
LIN {X 0,Y 255.504,Z 370.447,A -85,B 0,C 180,E1 -18620.502,E2 -18620.502} C_VEL
LIN {X 0,Y 254.829,Z 373.996,A -85,B 0,C 180,E1 -18623.148,E2 -18623.148} C_VEL
LIN {X 0,Y 254.479,Z 375.96,A -85,B 0,C 180,E1 -18625.248,E2 -18625.248} C_VEL
LIN {X 0,Y 254.302,Z 376.949,A -85,B 0,C 180,E1 -18626.832,E2 -18626.832} C_VEL
LIN {X 0,Y 254.114,Z 377.789,A -85,B 0,C 180,E1 -18630.001,E2 -18630.001} C_VEL
LIN {X 0,Y 254.147,Z 377.596,A -85,B 0,C 180,E1 -18631.585,E2 -18631.585} C_VEL
LIN {X 0,Y 254.3,Z 377.01,A -85,B 0,C 180,E1 -18633.169,E2 -18633.169} C_VEL
LIN {X 0,Y 254.473,Z 376.045,A -85,B 0,C 180,E1 -18634.753,E2 -18634.753} C_VEL
LIN {X 0,Y 254.829,Z 374.133,A -85,B 0,C 180,E1 -18636.852,E2 -18636.852} C_VEL
LIN {X 0,Y 255.48,Z 370.64,A -85,B 0,C 180,E1 -18639.501,E2 -18639.501} C_VEL
LIN {X 0,Y 256.465,Z 366.394,A -85,B 0,C 180,E1 -18641.861,E2 -18641.861} C_VEL
LIN {X 0,Y 258.061,Z 359.96,A -85,B 0,C 180,E1 -18644.591,E2 -18644.591} C_VEL
LIN {X 0,Y 259.703,Z 352.89,A -85,B 0,C 180,E1 -18646.913,E2 -18646.913} C_VEL
LIN {X 0,Y 261.851,Z 344.072,A -85,B 0,C 180,E1 -18649.196,E2 -18649.196} C_VEL
LIN {X 0,Y 263.801,Z 334.547,A -85,B 0,C 180,E1 -18651.18,E2 -18651.18} C_VEL
LIN {X 0,Y 265.559,Z 325.003,A -85,B 0,C 180,E1 -18652.772,E2 -18652.772} C_VEL
LIN {X 0,Y 267.442,Z 313.847,A -85,B 0,C 180,E1 -18654.243,E2 -18654.243} C_VEL
LIN {X 0,Y 268.98,Z 303.298,A -85,B 0,C 180,E1 -18655.332,E2 -18655.332} C_VEL
LIN {X 0,Y 270.423,Z 290.581,A -85,B 0,C 180,E1 -18656.324,E2 -18656.324} C_VEL
LIN {X 0,Y 271.391,Z 277.862,A -85,B 0,C 180,E1 -18657.001,E2 -18657.001} C_VEL
LIN {X 0,Y 272.218,Z 259.817,A -85,B 0,C 180,E1 -18657.536,E2 -18657.536} C_VEL
LIN {X 0,Y 273.719,Z 205.845,A -85,B 0,C 180,E1 -18658.947,E2 -18658.947} C_VEL
LIN {X 0,Y 266.996,Z 189.4,A -85,B 0,C 180,E1 -18660.258,E2 -18660.258} C_VEL
LIN {X 0,Y 259.93,Z 174.571,A -85,B 0,C 180,E1 -18661.651,E2 -18661.651} C_VEL
LIN {X 0,Y 256.299,Z 167.583,A -85,B 0,C 180,E1 -18662.384,E2 -18662.384} C_VEL
LIN {X 0,Y 256.079,Z 166.583,A -85,B 0,C 180,E1 -18662.76,E2 -18662.76} C_VEL
LIN {X 0,Y 256.081,Z 166.586,A -85,B 0,C 180,E1 -18665.193,E2 -18665.193} C_VEL
LIN {X 0,Y 256.117,Z 166.58,A -85,B 0,C 180,E1 -18667.271,E2 -18667.271} C_VEL
LIN {X 0,Y 256.032,Z 166.592,A -85,B 0,C 180,E1 -18672.171,E2 -18672.171} C_VEL
LIN {X 0,Y 256.023,Z 166.59,A -85,B 0,C 180,E1 -18676.664,E2 -18676.664} C_VEL
LIN {X 0,Y 256.067,Z 166.581,A -85,B 0,C 180,E1 -18680.857,E2 -18680.857} C_VEL
LIN {X 0,Y 256.126,Z 166.581,A -85,B 0,C 180,E1 -18682.866,E2 -18682.866} C_VEL
LIN {X 0,Y 256.067,Z 166.585,A -85,B 0,C 180,E1 -18686.707,E2 -18686.707} C_VEL
LIN {X 0,Y 256.055,Z 166.581,A -85,B 0,C 180,E1 -18690.393,E2 -18690.393} C_VEL
LIN {X 0,Y 256.134,Z 166.579,A -85,B 0,C 180,E1 -18694.888,E2 -18694.888} C_VEL
LIN {X 0,Y 256.149,Z 166.574,A -85,B 0,C 180,E1 -18699.103,E2 -18699.103} C_VEL
LIN {X 0,Y 256.213,Z 166.559,A -85,B 0,C 180,E1 -18704.079,E2 -18704.079} C_VEL
LIN {X 0,Y 256.287,Z 166.56,A -85,B 0,C 180,E1 -18708.933,E2 -18708.933} C_VEL
LIN {X 0,Y 256.467,Z 166.526,A -85,B 0,C 180,E1 -18712.125,E2 -18712.125} C_VEL
LIN {X 0,Y 256.447,Z 166.54,A -85,B 0,C 180,E1 -18716.858,E2 -18716.858} C_VEL
LIN {X 0,Y 256.574,Z 166.52,A -85,B 0,C 180,E1 -18717.814,E2 -18717.814} C_VEL
LIN {X 0,Y 256.034,Z 166.587,A -85,B 0,C 180,E1 -18719.124,E2 -18719.124} C_VEL
LIN {X 0,Y 254.435,Z 166.783,A -85,B 0,C 180,E1 -18720.409,E2 -18720.409} C_VEL
LIN {X 0,Y 250.489,Z 167.275,A -85,B 0,C 180,E1 -18722.991,E2 -18722.991} C_VEL
LIN {X 0,Y 249.35,Z 167.425,A -85,B 0,C 180,E1 -18724.343,E2 -18724.343} C_VEL
LIN {X 0,Y 249.252,Z 167.435,A -85,B 0,C 180,E1 -18724.802,E2 -18724.802} C_VEL
LIN {X 0,Y 249.402,Z 167.406,A -85,B 0,C 180,E1 -18728.1,E2 -18728.1} C_VEL
LIN {X 0,Y 249.214,Z 167.435,A -85,B 0,C 180,E1 -18731.385,E2 -18731.385} C_VEL
LIN {X 0,Y 249.151,Z 167.434,A -85,B 0,C 180,E1 -18736.45,E2 -18736.45} C_VEL
LIN {X 0,Y 249.042,Z 167.459,A -85,B 0,C 180,E1 -18741.522,E2 -18741.522} C_VEL
LIN {X 0,Y 249.047,Z 167.462,A -85,B 0,C 180,E1 -18745.441,E2 -18745.441} C_VEL
LIN {X 0,Y 249.033,Z 167.456,A -85,B 0,C 180,E1 -18748.972,E2 -18748.972} C_VEL
LIN {X 0,Y 249.028,Z 167.464,A -85,B 0,C 180,E1 -18752.426,E2 -18752.426} C_VEL
LIN {X 0,Y 249.023,Z 167.465,A -85,B 0,C 180,E1 -18756.347,E2 -18756.347} C_VEL
LIN {X 0,Y 248.979,Z 167.472,A -85,B 0,C 180,E1 -18760.483,E2 -18760.483} C_VEL
LIN {X 0,Y 248.962,Z 167.47,A -85,B 0,C 180,E1 -18764.889,E2 -18764.889} C_VEL
LIN {X 0,Y 248.98,Z 167.467,A -85,B 0,C 180,E1 -18767.355,E2 -18767.355} C_VEL
LIN {X 0,Y 249.064,Z 167.666,A -85,B 0,C 180,E1 -18770.909,E2 -18770.909} C_VEL
LIN {X 0,Y 251.11,Z 175.523,A -85,B 0,C 180,E1 -18774.257,E2 -18774.257} C_VEL
LIN {X 0,Y 252.741,Z 182.8,A -85,B 0,C 180,E1 -18777.134,E2 -18777.134} C_VEL
LIN {X 0,Y 260.868,Z 201.432,A -85,B 0,C 180,E1 -18778.857,E2 -18778.857} C_VEL
LIN {X 0,Y 262.459,Z 206.067,A -85,B 0,C 180,E1 -18779.209,E2 -18779.209} C_VEL
LIN {X 0,Y 265.885,Z 228.872,A -85,B 0,C 180,E1 -18780.339,E2 -18780.339} C_VEL
LIN {X 0,Y 266.642,Z 236.067,A -85,B 0,C 180,E1 -18780.648,E2 -18780.648} C_VEL
LIN {X 0,Y 264.775,Z 291.986,A -85,B 0,C 180,E1 -18782.16,E2 -18782.16} C_VEL
LIN {X 0,Y 263.629,Z 305.124,A -85,B 0,C 180,E1 -18782.783,E2 -18782.783} C_VEL
LIN {X 0,Y 262.11,Z 317.215,A -85,B 0,C 180,E1 -18783.634,E2 -18783.634} C_VEL
LIN {X 0,Y 260.203,Z 329.428,A -85,B 0,C 180,E1 -18784.823,E2 -18784.823} C_VEL
LIN {X 0,Y 258.012,Z 341.001,A -85,B 0,C 180,E1 -18786.31,E2 -18786.31} C_VEL
LIN {X 0,Y 255.788,Z 351.427,A -85,B 0,C 180,E1 -18788.015,E2 -18788.015} C_VEL
LIN {X 0,Y 253.921,Z 359.958,A -85,B 0,C 180,E1 -18789.758,E2 -18789.758} C_VEL
LIN {X 0,Y 252.278,Z 367.732,A -85,B 0,C 180,E1 -18791.704,E2 -18791.704} C_VEL
LIN {X 0,Y 250.4,Z 375.531,A -85,B 0,C 180,E1 -18794.118,E2 -18794.118} C_VEL
LIN {X 0,Y 248.641,Z 382.63,A -85,B 0,C 180,E1 -18796.93,E2 -18796.93} C_VEL
LIN {X 0,Y 247.784,Z 387.364,A -85,B 0,C 180,E1 -18799.375,E2 -18799.375} C_VEL
LIN {X 0,Y 247.197,Z 390.983,A -85,B 0,C 180,E1 -18801.827,E2 -18801.827} C_VEL
LIN {X 0,Y 246.976,Z 392.851,A -85,B 0,C 180,E1 -18803.463,E2 -18803.463} C_VEL
LIN {X 0,Y 246.883,Z 394.254,A -85,B 0,C 180,E1 -18805.1,E2 -18805.1} C_VEL
LIN {X 0,Y 246.898,Z 395.259,A -85,B 0,C 180,E1 -18806.736,E2 -18806.736} C_VEL
LIN {X 0,Y 246.977,Z 395.873,A -85,B 0,C 180,E1 -18808.369,E2 -18808.369} C_VEL
LIN {X 0,Y 247.028,Z 396.088,A -85,B 0,C 180,E1 -18809.999,E2 -18809.999} C_VEL
LIN {X 0,Y 246.977,Z 395.863,A -85,B 0,C 180,E1 -18811.63,E2 -18811.63} C_VEL
LIN {X 0,Y 246.898,Z 395.243,A -85,B 0,C 180,E1 -18813.263,E2 -18813.263} C_VEL
LIN {X 0,Y 246.882,Z 394.233,A -85,B 0,C 180,E1 -18814.898,E2 -18814.898} C_VEL
LIN {X 0,Y 246.981,Z 392.82,A -85,B 0,C 180,E1 -18816.535,E2 -18816.535} C_VEL
LIN {X 0,Y 247.395,Z 389.861,A -85,B 0,C 180,E1 -18818.988,E2 -18818.988} C_VEL
LIN {X 0,Y 248.052,Z 385.861,A -85,B 0,C 180,E1 -18821.438,E2 -18821.438} C_VEL
LIN {X 0,Y 249.349,Z 379.72,A -85,B 0,C 180,E1 -18824.277,E2 -18824.277} C_VEL
LIN {X 0,Y 250.889,Z 373.021,A -85,B 0,C 180,E1 -18826.685,E2 -18826.685} C_VEL
